LIN {X 0,Y 453.515,Z 483.113,A -85,B 0,C 180,E1 -8409.446,E2 -8409.446} C_VEL
LIN {X 0,Y 453.464,Z 483.111,A -85,B 0,C 180,E1 -8412.994,E2 -8412.994} C_VEL
LIN {X 0,Y 453.46,Z 483.124,A -85,B 0,C 180,E1 -8415.778,E2 -8415.778} C_VEL
LIN {X 0,Y 453.512,Z 483.122,A -85,B 0,C 180,E1 -8419.405,E2 -8419.405} C_VEL
LIN {X 0,Y 453.471,Z 483.115,A -85,B 0,C 180,E1 -8422.222,E2 -8422.222} C_VEL
LIN {X 0,Y 453.484,Z 483.123,A -85,B 0,C 180,E1 -8425.222,E2 -8425.222} C_VEL
LIN {X 0,Y 453.46,Z 483.119,A -85,B 0,C 180,E1 -8428.474,E2 -8428.474} C_VEL
LIN {X 0,Y 453.531,Z 483.104,A -85,B 0,C 180,E1 -8432.038,E2 -8432.038} C_VEL
LIN {X 0,Y 453.507,Z 483.119,A -85,B 0,C 180,E1 -8435.265,E2 -8435.265} C_VEL
LIN {X 0,Y 453.473,Z 483.112,A -85,B 0,C 180,E1 -8438.414,E2 -8438.414} C_VEL
LIN {X 0,Y 453.514,Z 483.11,A -85,B 0,C 180,E1 -8441.008,E2 -8441.008} C_VEL
LIN {X 0,Y 453.561,Z 483.108,A -85,B 0,C 180,E1 -8443.879,E2 -8443.879} C_VEL
LIN {X 0,Y 453.555,Z 483.102,A -85,B 0,C 180,E1 -8447.471,E2 -8447.471} C_VEL
LIN {X 0,Y 453.584,Z 483.109,A -85,B 0,C 180,E1 -8451.086,E2 -8451.086} C_VEL
LIN {X 0,Y 453.669,Z 483.082,A -85,B 0,C 180,E1 -8453.774,E2 -8453.774} C_VEL
LIN {X 0,Y 453.757,Z 483.086,A -85,B 0,C 180,E1 -8457.336,E2 -8457.336} C_VEL
LIN {X 0,Y 453.814,Z 483.072,A -85,B 0,C 180,E1 -8460,E2 -8460} C_VEL
LIN {X 0,Y 453.757,Z 483.069,A -85,B 0,C 180,E1 -8462.663,E2 -8462.663} C_VEL
LIN {X 0,Y 453.667,Z 483.095,A -85,B 0,C 180,E1 -8466.225,E2 -8466.225} C_VEL
LIN {X 0,Y 453.583,Z 483.099,A -85,B 0,C 180,E1 -8468.913,E2 -8468.913} C_VEL
LIN {X 0,Y 453.554,Z 483.108,A -85,B 0,C 180,E1 -8472.529,E2 -8472.529} C_VEL
LIN {X 0,Y 453.535,Z 483.104,A -85,B 0,C 180,E1 -8476.196,E2 -8476.196} C_VEL
LIN {X 0,Y 453.51,Z 483.11,A -85,B 0,C 180,E1 -8479.041,E2 -8479.041} C_VEL
LIN {X 0,Y 453.466,Z 483.122,A -85,B 0,C 180,E1 -8481.836,E2 -8481.836} C_VEL
LIN {X 0,Y 453.504,Z 483.105,A -85,B 0,C 180,E1 -8484.734,E2 -8484.734} C_VEL
LIN {X 0,Y 453.529,Z 483.115,A -85,B 0,C 180,E1 -8487.961,E2 -8487.961} C_VEL
LIN {X 0,Y 453.474,Z 483.109,A -85,B 0,C 180,E1 -8490.759,E2 -8490.759} C_VEL
LIN {X 0,Y 453.469,Z 483.123,A -85,B 0,C 180,E1 -8493.913,E2 -8493.913} C_VEL
LIN {X 0,Y 453.462,Z 483.119,A -85,B 0,C 180,E1 -8497.188,E2 -8497.188} C_VEL
LIN {X 0,Y 453.508,Z 483.121,A -85,B 0,C 180,E1 -8499.447,E2 -8499.447} C_VEL
LIN {X 0,Y 453.484,Z 483.12,A -85,B 0,C 180,E1 -8502.992,E2 -8502.992} C_VEL
LIN {X 0,Y 453.469,Z 483.104,A -85,B 0,C 180,E1 -8505.781,E2 -8505.781} C_VEL
LIN {X 0,Y 453.49,Z 483.109,A -85,B 0,C 180,E1 -8508.212,E2 -8508.212} C_VEL
LIN {X 0,Y 453.528,Z 483.114,A -85,B 0,C 180,E1 -8510.787,E2 -8510.787} C_VEL
LIN {X 0,Y 453.45,Z 483.113,A -85,B 0,C 180,E1 -8513.918,E2 -8513.918} C_VEL
LIN {X 0,Y 453.477,Z 483.122,A -85,B 0,C 180,E1 -8517.152,E2 -8517.152} C_VEL
LIN {X 0,Y 453.508,Z 483.12,A -85,B 0,C 180,E1 -8520.271,E2 -8520.271} C_VEL
LIN {X 0,Y 453.504,Z 483.12,A -85,B 0,C 180,E1 -8523.294,E2 -8523.294} C_VEL
LIN {X 0,Y 453.499,Z 483.122,A -85,B 0,C 180,E1 -8526.239,E2 -8526.239} C_VEL
LIN {X 0,Y 453.478,Z 483.122,A -85,B 0,C 180,E1 -8529.118,E2 -8529.118} C_VEL
LIN {X 0,Y 453.507,Z 483.123,A -85,B 0,C 180,E1 -8531.945,E2 -8531.945} C_VEL
LIN {X 0,Y 453.535,Z 483.116,A -85,B 0,C 180,E1 -8534.727,E2 -8534.727} C_VEL
LIN {X 0,Y 453.556,Z 483.115,A -85,B 0,C 180,E1 -8538.379,E2 -8538.379} C_VEL
LIN {X 0,Y 453.648,Z 483.104,A -85,B 0,C 180,E1 -8541.985,E2 -8541.985} C_VEL
LIN {X 0,Y 453.633,Z 483.102,A -85,B 0,C 180,E1 -8543.101,E2 -8543.101} C_VEL
LIN {X 0,Y 452.948,Z 483.192,A -85,B 0,C 180,E1 -8543.841,E2 -8543.841} C_VEL
LIN {X 0,Y 450,Z 483.556,A -85,B 0,C 180,E1 -8545.043,E2 -8545.043} C_VEL
LIN {X 0,Y 447.578,Z 483.861,A -85,B 0,C 180,E1 -8546.012,E2 -8546.012} C_VEL
LIN {X 0,Y 446.643,Z 483.975,A -85,B 0,C 180,E1 -8546.762,E2 -8546.762} C_VEL
LIN {X 0,Y 446.623,Z 483.977,A -85,B 0,C 180,E1 -8547.016,E2 -8547.016} C_VEL
LIN {X 0,Y 446.791,Z 483.959,A -85,B 0,C 180,E1 -8550,E2 -8550} C_VEL
LIN {X 0,Y 446.706,Z 483.968,A -85,B 0,C 180,E1 -8552.705,E2 -8552.705} C_VEL
LIN {X 0,Y 446.643,Z 483.977,A -85,B 0,C 180,E1 -8556.324,E2 -8556.324} C_VEL
LIN {X 0,Y 446.534,Z 483.987,A -85,B 0,C 180,E1 -8559.055,E2 -8559.055} C_VEL
LIN {X 0,Y 446.517,Z 483.99,A -85,B 0,C 180,E1 -8562.73,E2 -8562.73} C_VEL
LIN {X 0,Y 446.492,Z 483.996,A -85,B 0,C 180,E1 -8566.228,E2 -8566.228} C_VEL
LIN {X 0,Y 446.465,Z 483.997,A -85,B 0,C 180,E1 -8569.303,E2 -8569.303} C_VEL
LIN {X 0,Y 446.414,Z 484.005,A -85,B 0,C 180,E1 -8572.199,E2 -8572.199} C_VEL
LIN {X 0,Y 446.452,Z 483.997,A -85,B 0,C 180,E1 -8575.152,E2 -8575.152} C_VEL
LIN {X 0,Y 446.479,Z 483.998,A -85,B 0,C 180,E1 -8578.178,E2 -8578.178} C_VEL
LIN {X 0,Y 446.414,Z 484.001,A -85,B 0,C 180,E1 -8581.3,E2 -8581.3} C_VEL
LIN {X 0,Y 446.424,Z 484,A -85,B 0,C 180,E1 -8584.523,E2 -8584.523} C_VEL
LIN {X 0,Y 446.431,Z 483.991,A -85,B 0,C 180,E1 -8588.083,E2 -8588.083} C_VEL
LIN {X 0,Y 446.44,Z 483.993,A -85,B 0,C 180,E1 -8590.92,E2 -8590.92} C_VEL
LIN {X 0,Y 446.437,Z 483.973,A -85,B 0,C 180,E1 -8593.84,E2 -8593.84} C_VEL
LIN {X 0,Y 446.439,Z 484.003,A -85,B 0,C 180,E1 -8596.397,E2 -8596.397} C_VEL
LIN {X 0,Y 446.443,Z 483.991,A -85,B 0,C 180,E1 -8599.803,E2 -8599.803} C_VEL
LIN {X 0,Y 446.419,Z 484.005,A -85,B 0,C 180,E1 -8602.123,E2 -8602.123} C_VEL
LIN {X 0,Y 446.421,Z 483.996,A -85,B 0,C 180,E1 -8605.477,E2 -8605.477} C_VEL
LIN {X 0,Y 446.41,Z 483.992,A -85,B 0,C 180,E1 -8608.7,E2 -8608.7} C_VEL
LIN {X 0,Y 446.475,Z 483.992,A -85,B 0,C 180,E1 -8611.821,E2 -8611.821} C_VEL
LIN {X 0,Y 446.448,Z 483.986,A -85,B 0,C 180,E1 -8614.848,E2 -8614.848} C_VEL
LIN {X 0,Y 446.438,Z 483.999,A -85,B 0,C 180,E1 -8618.245,E2 -8618.245} C_VEL
LIN {X 0,Y 446.448,Z 483.988,A -85,B 0,C 180,E1 -8621.649,E2 -8621.649} C_VEL
LIN {X 0,Y 446.498,Z 483.989,A -85,B 0,C 180,E1 -8624.48,E2 -8624.48} C_VEL
LIN {X 0,Y 446.509,Z 483.988,A -85,B 0,C 180,E1 -8628.193,E2 -8628.193} C_VEL
LIN {X 0,Y 446.591,Z 483.97,A -85,B 0,C 180,E1 -8631.858,E2 -8631.858} C_VEL
LIN {X 0,Y 446.643,Z 483.973,A -85,B 0,C 180,E1 -8634.583,E2 -8634.583} C_VEL
LIN {X 0,Y 446.701,Z 483.948,A -85,B 0,C 180,E1 -8637.295,E2 -8637.295} C_VEL
LIN {X 0,Y 446.784,Z 483.947,A -85,B 0,C 180,E1 -8640,E2 -8640} C_VEL
LIN {X 0,Y 446.701,Z 483.964,A -85,B 0,C 180,E1 -8642.706,E2 -8642.706} C_VEL
LIN {X 0,Y 446.638,Z 483.958,A -85,B 0,C 180,E1 -8646.324,E2 -8646.324} C_VEL
LIN {X 0,Y 446.53,Z 483.987,A -85,B 0,C 180,E1 -8649.056,E2 -8649.056} C_VEL
LIN {X 0,Y 446.513,Z 483.976,A -85,B 0,C 180,E1 -8652.73,E2 -8652.73} C_VEL
LIN {X 0,Y 446.482,Z 483.994,A -85,B 0,C 180,E1 -8656.46,E2 -8656.46} C_VEL
LIN {X 0,Y 446.462,Z 483.986,A -85,B 0,C 180,E1 -8659.304,E2 -8659.304} C_VEL
LIN {X 0,Y 446.411,Z 483.994,A -85,B 0,C 180,E1 -8662.2,E2 -8662.2} C_VEL
LIN {X 0,Y 446.451,Z 483.993,A -85,B 0,C 180,E1 -8665.153,E2 -8665.153} C_VEL
LIN {X 0,Y 446.478,Z 483.984,A -85,B 0,C 180,E1 -8668.179,E2 -8668.179} C_VEL
LIN {X 0,Y 446.414,Z 483.997,A -85,B 0,C 180,E1 -8671.776,E2 -8671.776} C_VEL
LIN {X 0,Y 446.425,Z 483.998,A -85,B 0,C 180,E1 -8674.524,E2 -8674.524} C_VEL
LIN {X 0,Y 446.431,Z 483.992,A -85,B 0,C 180,E1 -8678.084,E2 -8678.084} C_VEL
LIN {X 0,Y 446.439,Z 483.998,A -85,B 0,C 180,E1 -8680.921,E2 -8680.921} C_VEL
LIN {X 0,Y 446.396,Z 484.003,A -85,B 0,C 180,E1 -8683.847,E2 -8683.847} C_VEL
LIN {X 0,Y 446.417,Z 483.989,A -85,B 0,C 180,E1 -8686.401,E2 -8686.401} C_VEL
LIN {X 0,Y 446.449,Z 483.996,A -85,B 0,C 180,E1 -8689.804,E2 -8689.804} C_VEL
LIN {X 0,Y 446.407,Z 483.973,A -85,B 0,C 180,E1 -8692.122,E2 -8692.122} C_VEL
LIN {X 0,Y 446.428,Z 483.989,A -85,B 0,C 180,E1 -8695.478,E2 -8695.478} C_VEL
LIN {X 0,Y 446.417,Z 483.974,A -85,B 0,C 180,E1 -8698.701,E2 -8698.701} C_VEL
LIN {X 0,Y 446.476,Z 484.115,A -85,B 0,C 180,E1 -8699.755,E2 -8699.755} C_VEL
LIN {X 0,Y 448.83,Z 495.487,A -85,B 0,C 180,E1 -8702.489,E2 -8702.489} C_VEL
LIN {X 0,Y 449.538,Z 500.19,A -85,B 0,C 180,E1 -8703.541,E2 -8703.541} C_VEL
LIN {X 0,Y 448.777,Z 514.196,A -85,B 0,C 180,E1 -8706.464,E2 -8706.464} C_VEL
LIN {X 0,Y 448.217,Z 523.143,A -85,B 0,C 180,E1 -8708.318,E2 -8708.318} C_VEL
LIN {X 0,Y 449.163,Z 527.943,A -85,B 0,C 180,E1 -8708.491,E2 -8708.491} C_VEL
LIN {X 0,Y 453.386,Z 549.291,A -85,B 0,C 180,E1 -8709.054,E2 -8709.054} C_VEL
LIN {X 0,Y 452.142,Z 657.267,A -85,B 0,C 180,E1 -8710.802,E2 -8710.802} C_VEL
LIN {X 0,Y 451.794,Z 668.666,A -85,B 0,C 180,E1 -8711.081,E2 -8711.081} C_VEL
LIN {X 0,Y 451.343,Z 679.209,A -85,B 0,C 180,E1 -8711.444,E2 -8711.444} C_VEL
LIN {X 0,Y 450.892,Z 689.76,A -85,B 0,C 180,E1 -8711.921,E2 -8711.921} C_VEL
LIN {X 0,Y 450.291,Z 700.274,A -85,B 0,C 180,E1 -8712.511,E2 -8712.511} C_VEL
LIN {X 0,Y 449.69,Z 710.266,A -85,B 0,C 180,E1 -8713.195,E2 -8713.195} C_VEL
LIN {X 0,Y 449.012,Z 719.993,A -85,B 0,C 180,E1 -8713.987,E2 -8713.987} C_VEL
LIN {X 0,Y 448.336,Z 729.416,A -85,B 0,C 180,E1 -8714.894,E2 -8714.894} C_VEL
LIN {X 0,Y 447.671,Z 738.441,A -85,B 0,C 180,E1 -8715.917,E2 -8715.917} C_VEL
LIN {X 0,Y 447.112,Z 746.926,A -85,B 0,C 180,E1 -8717.049,E2 -8717.049} C_VEL
LIN {X 0,Y 446.683,Z 754.285,A -85,B 0,C 180,E1 -8718.198,E2 -8718.198} C_VEL
LIN {X 0,Y 446.237,Z 760.559,A -85,B 0,C 180,E1 -8719.336,E2 -8719.336} C_VEL
LIN {X 0,Y 445.953,Z 765.962,A -85,B 0,C 180,E1 -8720.475,E2 -8720.475} C_VEL
LIN {X 0,Y 445.697,Z 771.394,A -85,B 0,C 180,E1 -8721.841,E2 -8721.841} C_VEL
LIN {X 0,Y 445.57,Z 775.838,A -85,B 0,C 180,E1 -8723.207,E2 -8723.207} C_VEL
LIN {X 0,Y 445.476,Z 779.378,A -85,B 0,C 180,E1 -8724.568,E2 -8724.568} C_VEL
LIN {X 0,Y 445.395,Z 781.314,A -85,B 0,C 180,E1 -8725.475,E2 -8725.475} C_VEL
LIN {X 0,Y 445.429,Z 783.994,A -85,B 0,C 180,E1 -8727.287,E2 -8727.287} C_VEL
LIN {X 0,Y 445.336,Z 785.278,A -85,B 0,C 180,E1 -8729.096,E2 -8729.096} C_VEL
LIN {X 0,Y 445.341,Z 785.529,A -85,B 0,C 180,E1 -8730,E2 -8730} C_VEL
LIN {X 0,Y 445.353,Z 784.807,A -85,B 0,C 180,E1 -8731.809,E2 -8731.809} C_VEL
LIN {X 0,Y 445.429,Z 783.994,A -85,B 0,C 180,E1 -8732.713,E2 -8732.713} C_VEL
LIN {X 0,Y 445.395,Z 781.314,A -85,B 0,C 180,E1 -8734.525,E2 -8734.525} C_VEL
LIN {X 0,Y 445.529,Z 776.974,A -85,B 0,C 180,E1 -8736.385,E2 -8736.385} C_VEL
LIN {X 0,Y 445.621,Z 772.972,A -85,B 0,C 180,E1 -8737.704,E2 -8737.704} C_VEL
LIN {X 0,Y 445.884,Z 767.876,A -85,B 0,C 180,E1 -8739.069,E2 -8739.069} C_VEL
LIN {X 0,Y 446.179,Z 761.697,A -85,B 0,C 180,E1 -8740.436,E2 -8740.436} C_VEL
LIN {X 0,Y 446.605,Z 755.623,A -85,B 0,C 180,E1 -8741.574,E2 -8741.574} C_VEL
LIN {X 0,Y 447.018,Z 748.545,A -85,B 0,C 180,E1 -8742.715,E2 -8742.715} C_VEL
LIN {X 0,Y 447.442,Z 742.08,A -85,B 0,C 180,E1 -8743.627,E2 -8743.627} C_VEL
LIN {X 0,Y 448.128,Z 732.597,A -85,B 0,C 180,E1 -8744.764,E2 -8744.764} C_VEL
LIN {X 0,Y 448.713,Z 723.714,A -85,B 0,C 180,E1 -8745.675,E2 -8745.675} C_VEL
LIN {X 0,Y 449.406,Z 714.661,A -85,B 0,C 180,E1 -8746.466,E2 -8746.466} C_VEL
LIN {X 0,Y 450.11,Z 703.851,A -85,B 0,C 180,E1 -8747.257,E2 -8747.257} C_VEL
LIN {X 0,Y 450.666,Z 694.13,A -85,B 0,C 180,E1 -8747.85,E2 -8747.85} C_VEL
LIN {X 0,Y 451.166,Z 683.291,A -85,B 0,C 180,E1 -8748.387,E2 -8748.387} C_VEL
LIN {X 0,Y 451.69,Z 671.402,A -85,B 0,C 180,E1 -8748.835,E2 -8748.835} C_VEL
LIN {X 0,Y 452.062,Z 659.986,A -85,B 0,C 180,E1 -8749.143,E2 -8749.143} C_VEL
LIN {X 0,Y 452.545,Z 631.666,A -85,B 0,C 180,E1 -8749.623,E2 -8749.623} C_VEL
LIN {X 0,Y 453.344,Z 548.908,A -85,B 0,C 180,E1 -8750.955,E2 -8750.955} C_VEL
LIN {X 0,Y 448.23,Z 523.43,A -85,B 0,C 180,E1 -8751.653,E2 -8751.653} C_VEL
LIN {X 0,Y 448.295,Z 522.142,A -85,B 0,C 180,E1 -8751.859,E2 -8751.859} C_VEL
LIN {X 0,Y 449.213,Z 507.408,A -85,B 0,C 180,E1 -8754.987,E2 -8754.987} C_VEL
LIN {X 0,Y 449.593,Z 500.365,A -85,B 0,C 180,E1 -8756.455,E2 -8756.455} C_VEL
LIN {X 0,Y 448.145,Z 491.791,A -85,B 0,C 180,E1 -8758.378,E2 -8758.378} C_VEL
LIN {X 0,Y 446.476,Z 484.118,A -85,B 0,C 180,E1 -8760.245,E2 -8760.245} C_VEL
LIN {X 0,Y 446.444,Z 484.003,A -85,B 0,C 180,E1 -8763.453,E2 -8763.453} C_VEL
LIN {X 0,Y 446.399,Z 483.96,A -85,B 0,C 180,E1 -8766.745,E2 -8766.745} C_VEL
LIN {X 0,Y 446.476,Z 483.991,A -85,B 0,C 180,E1 -8769.528,E2 -8769.528} C_VEL
LIN {X 0,Y 446.429,Z 483.99,A -85,B 0,C 180,E1 -8772.603,E2 -8772.603} C_VEL
LIN {X 0,Y 446.45,Z 483.993,A -85,B 0,C 180,E1 -8775.103,E2 -8775.103} C_VEL
LIN {X 0,Y 446.431,Z 483.994,A -85,B 0,C 180,E1 -8778.609,E2 -8778.609} C_VEL
LIN {X 0,Y 446.468,Z 483.997,A -85,B 0,C 180,E1 -8780.975,E2 -8780.975} C_VEL
LIN {X 0,Y 446.416,Z 483.999,A -85,B 0,C 180,E1 -8784.373,E2 -8784.373} C_VEL
LIN {X 0,Y 446.417,Z 483.998,A -85,B 0,C 180,E1 -8787.638,E2 -8787.638} C_VEL
LIN {X 0,Y 446.443,Z 483.997,A -85,B 0,C 180,E1 -8790.79,E2 -8790.79} C_VEL
LIN {X 0,Y 446.471,Z 483.991,A -85,B 0,C 180,E1 -8793.848,E2 -8793.848} C_VEL
LIN {X 0,Y 446.422,Z 483.999,A -85,B 0,C 180,E1 -8796.823,E2 -8796.823} C_VEL
LIN {X 0,Y 446.437,Z 483.989,A -85,B 0,C 180,E1 -8799.736,E2 -8799.736} C_VEL
LIN {X 0,Y 446.456,Z 483.994,A -85,B 0,C 180,E1 -8802.596,E2 -8802.596} C_VEL
LIN {X 0,Y 446.461,Z 483.986,A -85,B 0,C 180,E1 -8805.412,E2 -8805.412} C_VEL
LIN {X 0,Y 446.509,Z 483.984,A -85,B 0,C 180,E1 -8808.192,E2 -8808.192} C_VEL
LIN {X 0,Y 446.592,Z 483.975,A -85,B 0,C 180,E1 -8811.857,E2 -8811.857} C_VEL
LIN {X 0,Y 446.637,Z 483.954,A -85,B 0,C 180,E1 -8814.582,E2 -8814.582} C_VEL
LIN {X 0,Y 446.701,Z 483.964,A -85,B 0,C 180,E1 -8817.294,E2 -8817.294} C_VEL
LIN {X 0,Y 446.784,Z 483.947,A -85,B 0,C 180,E1 -8820,E2 -8820} C_VEL
LIN {X 0,Y 446.701,Z 483.948,A -85,B 0,C 180,E1 -8822.705,E2 -8822.705} C_VEL
LIN {X 0,Y 446.637,Z 483.97,A -85,B 0,C 180,E1 -8826.323,E2 -8826.323} C_VEL
LIN {X 0,Y 446.529,Z 483.978,A -85,B 0,C 180,E1 -8829.055,E2 -8829.055} C_VEL
LIN {X 0,Y 446.512,Z 483.986,A -85,B 0,C 180,E1 -8832.73,E2 -8832.73} C_VEL
LIN {X 0,Y 446.486,Z 483.981,A -85,B 0,C 180,E1 -8836.228,E2 -8836.228} C_VEL
LIN {X 0,Y 446.46,Z 483.99,A -85,B 0,C 180,E1 -8839.303,E2 -8839.303} C_VEL
LIN {X 0,Y 446.408,Z 483.998,A -85,B 0,C 180,E1 -8842.2,E2 -8842.2} C_VEL
LIN {X 0,Y 446.448,Z 483.986,A -85,B 0,C 180,E1 -8845.152,E2 -8845.152} C_VEL
LIN {X 0,Y 446.475,Z 483.992,A -85,B 0,C 180,E1 -8848.179,E2 -8848.179} C_VEL
LIN {X 0,Y 446.41,Z 483.992,A -85,B 0,C 180,E1 -8851.3,E2 -8851.3} C_VEL
LIN {X 0,Y 446.421,Z 483.996,A -85,B 0,C 180,E1 -8854.523,E2 -8854.523} C_VEL
LIN {X 0,Y 446.422,Z 484.002,A -85,B 0,C 180,E1 -8858.082,E2 -8858.082} C_VEL
LIN {X 0,Y 446.422,Z 483.991,A -85,B 0,C 180,E1 -8860.918,E2 -8860.918} C_VEL
LIN {X 0,Y 446.437,Z 483.999,A -85,B 0,C 180,E1 -8863.841,E2 -8863.841} C_VEL
LIN {X 0,Y 446.439,Z 483.97,A -85,B 0,C 180,E1 -8866.397,E2 -8866.397} C_VEL
LIN {X 0,Y 446.463,Z 483.998,A -85,B 0,C 180,E1 -8869.805,E2 -8869.805} C_VEL
LIN {X 0,Y 446.428,Z 483.989,A -85,B 0,C 180,E1 -8872.124,E2 -8872.124} C_VEL
LIN {X 0,Y 446.424,Z 484,A -85,B 0,C 180,E1 -8875.477,E2 -8875.477} C_VEL
LIN {X 0,Y 446.414,Z 484.001,A -85,B 0,C 180,E1 -8878.7,E2 -8878.7} C_VEL
LIN {X 0,Y 446.479,Z 483.998,A -85,B 0,C 180,E1 -8881.822,E2 -8881.822} C_VEL
LIN {X 0,Y 446.452,Z 483.997,A -85,B 0,C 180,E1 -8884.848,E2 -8884.848} C_VEL
LIN {X 0,Y 446.443,Z 484.001,A -85,B 0,C 180,E1 -8888.245,E2 -8888.245} C_VEL
LIN {X 0,Y 446.453,Z 484,A -85,B 0,C 180,E1 -8891.649,E2 -8891.649} C_VEL
LIN {X 0,Y 446.503,Z 483.993,A -85,B 0,C 180,E1 -8894.48,E2 -8894.48} C_VEL
LIN {X 0,Y 446.514,Z 483.993,A -85,B 0,C 180,E1 -8898.193,E2 -8898.193} C_VEL
LIN {X 0,Y 446.596,Z 483.982,A -85,B 0,C 180,E1 -8901.858,E2 -8901.858} C_VEL
LIN {X 0,Y 446.642,Z 483.975,A -85,B 0,C 180,E1 -8904.583,E2 -8904.583} C_VEL
LIN {X 0,Y 446.623,Z 483.977,A -85,B 0,C 180,E1 -8907.016,E2 -8907.016} C_VEL
LIN {X 0,Y 446.106,Z 484.044,A -85,B 0,C 180,E1 -8907.769,E2 -8907.769} C_VEL
LIN {X 0,Y 443.288,Z 484.397,A -85,B 0,C 180,E1 -8908.992,E2 -8908.992} C_VEL
LIN {X 0,Y 440.8,Z 484.706,A -85,B 0,C 180,E1 -8909.979,E2 -8909.979} C_VEL
LIN {X 0,Y 439.712,Z 484.84,A -85,B 0,C 180,E1 -8910.742,E2 -8910.742} C_VEL
LIN {X 0,Y 439.618,Z 484.85,A -85,B 0,C 180,E1 -8911.001,E2 -8911.001} C_VEL
LIN {X 0,Y 439.652,Z 484.847,A -85,B 0,C 180,E1 -8912.749,E2 -8912.749} C_VEL
LIN {X 0,Y 439.614,Z 484.852,A -85,B 0,C 180,E1 -8916.425,E2 -8916.425} C_VEL
LIN {X 0,Y 439.496,Z 484.864,A -85,B 0,C 180,E1 -8919.201,E2 -8919.201} C_VEL
LIN {X 0,Y 439.461,Z 484.869,A -85,B 0,C 180,E1 -8922.937,E2 -8922.937} C_VEL
LIN {X 0,Y 439.443,Z 484.873,A -85,B 0,C 180,E1 -8926.349,E2 -8926.349} C_VEL
LIN {X 0,Y 439.398,Z 484.878,A -85,B 0,C 180,E1 -8929.626,E2 -8929.626} C_VEL
LIN {X 0,Y 439.361,Z 484.882,A -85,B 0,C 180,E1 -8932.575,E2 -8932.575} C_VEL
LIN {X 0,Y 439.4,Z 484.878,A -85,B 0,C 180,E1 -8935.585,E2 -8935.585} C_VEL
LIN {X 0,Y 439.419,Z 484.875,A -85,B 0,C 180,E1 -8938.673,E2 -8938.673} C_VEL
LIN {X 0,Y 439.369,Z 484.883,A -85,B 0,C 180,E1 -8941.86,E2 -8941.86} C_VEL
LIN {X 0,Y 439.394,Z 484.872,A -85,B 0,C 180,E1 -8945.155,E2 -8945.155} C_VEL
LIN {X 0,Y 439.393,Z 484.877,A -85,B 0,C 180,E1 -8948.593,E2 -8948.593} C_VEL
LIN {X 0,Y 439.397,Z 484.869,A -85,B 0,C 180,E1 -8951.259,E2 -8951.259} C_VEL
LIN {X 0,Y 439.402,Z 484.865,A -85,B 0,C 180,E1 -8954.728,E2 -8954.728} C_VEL
LIN {X 0,Y 439.403,Z 484.876,A -85,B 0,C 180,E1 -8957.797,E2 -8957.797} C_VEL
LIN {X 0,Y 439.428,Z 484.87,A -85,B 0,C 180,E1 -8960.228,E2 -8960.228} C_VEL
LIN {X 0,Y 439.368,Z 484.874,A -85,B 0,C 180,E1 -8963.713,E2 -8963.713} C_VEL
LIN {X 0,Y 439.366,Z 484.877,A -85,B 0,C 180,E1 -8967.054,E2 -8967.054} C_VEL
LIN {X 0,Y 439.387,Z 484.869,A -85,B 0,C 180,E1 -8970.275,E2 -8970.275} C_VEL
LIN {X 0,Y 439.424,Z 484.869,A -85,B 0,C 180,E1 -8973.589,E2 -8973.589} C_VEL
LIN {X 0,Y 439.377,Z 484.869,A -85,B 0,C 180,E1 -8976.43,E2 -8976.43} C_VEL
LIN {X 0,Y 439.379,Z 484.875,A -85,B 0,C 180,E1 -8979.397,E2 -8979.397} C_VEL
LIN {X 0,Y 439.422,Z 484.861,A -85,B 0,C 180,E1 -8982.31,E2 -8982.31} C_VEL
LIN {X 0,Y 439.437,Z 484.868,A -85,B 0,C 180,E1 -8985.174,E2 -8985.174} C_VEL
LIN {X 0,Y 439.475,Z 484.865,A -85,B 0,C 180,E1 -8988.002,E2 -8988.002} C_VEL
LIN {X 0,Y 439.539,Z 484.847,A -85,B 0,C 180,E1 -8991.727,E2 -8991.727} C_VEL
LIN {X 0,Y 439.618,Z 484.85,A -85,B 0,C 180,E1 -8994.496,E2 -8994.496} C_VEL
LIN {X 0,Y 439.627,Z 484.83,A -85,B 0,C 180,E1 -8998.168,E2 -8998.168} C_VEL
LIN {X 0,Y 439.754,Z 484.823,A -85,B 0,C 180,E1 -9000,E2 -9000} C_VEL
LIN {X 0,Y 439.648,Z 484.842,A -85,B 0,C 180,E1 -9002.749,E2 -9002.749} C_VEL
LIN {X 0,Y 439.609,Z 484.834,A -85,B 0,C 180,E1 -9006.426,E2 -9006.426} C_VEL
LIN {X 0,Y 439.492,Z 484.862,A -85,B 0,C 180,E1 -9009.202,E2 -9009.202} C_VEL
LIN {X 0,Y 439.458,Z 484.852,A -85,B 0,C 180,E1 -9012.938,E2 -9012.938} C_VEL
LIN {X 0,Y 439.439,Z 484.869,A -85,B 0,C 180,E1 -9016.349,E2 -9016.349} C_VEL
LIN {X 0,Y 439.395,Z 484.866,A -85,B 0,C 180,E1 -9019.627,E2 -9019.627} C_VEL
LIN {X 0,Y 439.358,Z 484.878,A -85,B 0,C 180,E1 -9022.576,E2 -9022.576} C_VEL
LIN {X 0,Y 439.399,Z 484.869,A -85,B 0,C 180,E1 -9025.586,E2 -9025.586} C_VEL
LIN {X 0,Y 439.411,Z 484.871,A -85,B 0,C 180,E1 -9028.674,E2 -9028.674} C_VEL
LIN {X 0,Y 439.365,Z 484.876,A -85,B 0,C 180,E1 -9032.031,E2 -9032.031} C_VEL
LIN {X 0,Y 439.391,Z 484.875,A -85,B 0,C 180,E1 -9035.342,E2 -9035.342} C_VEL
LIN {X 0,Y 439.392,Z 484.873,A -85,B 0,C 180,E1 -9038.594,E2 -9038.594} C_VEL
LIN {X 0,Y 439.394,Z 484.872,A -85,B 0,C 180,E1 -9041.259,E2 -9041.259} C_VEL
LIN {X 0,Y 439.398,Z 484.875,A -85,B 0,C 180,E1 -9044.73,E2 -9044.73} C_VEL
LIN {X 0,Y 439.395,Z 484.868,A -85,B 0,C 180,E1 -9047.797,E2 -9047.797} C_VEL
LIN {X 0,Y 439.434,Z 484.872,A -85,B 0,C 180,E1 -9050.229,E2 -9050.229} C_VEL
LIN {X 0,Y 439.371,Z 484.834,A -85,B 0,C 180,E1 -9053.714,E2 -9053.714} C_VEL
LIN {X 0,Y 439.372,Z 484.878,A -85,B 0,C 180,E1 -9057.055,E2 -9057.055} C_VEL
LIN {X 0,Y 439.439,Z 484.948,A -85,B 0,C 180,E1 -9059.442,E2 -9059.442} C_VEL
LIN {X 0,Y 441.81,Z 496.456,A -85,B 0,C 180,E1 -9062.272,E2 -9062.272} C_VEL
LIN {X 0,Y 442.632,Z 502.334,A -85,B 0,C 180,E1 -9063.604,E2 -9063.604} C_VEL
LIN {X 0,Y 441.67,Z 517.613,A -85,B 0,C 180,E1 -9066.832,E2 -9066.832} C_VEL
LIN {X 0,Y 441.34,Z 522.992,A -85,B 0,C 180,E1 -9067.97,E2 -9067.97} C_VEL
LIN {X 0,Y 442.627,Z 529.447,A -85,B 0,C 180,E1 -9068.186,E2 -9068.186} C_VEL
LIN {X 0,Y 446.778,Z 550.731,A -85,B 0,C 180,E1 -9068.757,E2 -9068.757} C_VEL
LIN {X 0,Y 445.406,Z 658.429,A -85,B 0,C 180,E1 -9070.53,E2 -9070.53} C_VEL
LIN {X 0,Y 445.047,Z 669.38,A -85,B 0,C 180,E1 -9070.813,E2 -9070.813} C_VEL
LIN {X 0,Y 444.546,Z 680.371,A -85,B 0,C 180,E1 -9071.209,E2 -9071.209} C_VEL
LIN {X 0,Y 444.096,Z 690.242,A -85,B 0,C 180,E1 -9071.672,E2 -9071.672} C_VEL
LIN {X 0,Y 443.489,Z 700.483,A -85,B 0,C 180,E1 -9072.262,E2 -9072.262} C_VEL
LIN {X 0,Y 442.848,Z 710.066,A -85,B 0,C 180,E1 -9072.927,E2 -9072.927} C_VEL
LIN {X 0,Y 442.164,Z 719.794,A -85,B 0,C 180,E1 -9073.732,E2 -9073.732} C_VEL
LIN {X 0,Y 441.467,Z 729.217,A -85,B 0,C 180,E1 -9074.653,E2 -9074.653} C_VEL
LIN {X 0,Y 440.753,Z 738.242,A -85,B 0,C 180,E1 -9075.691,E2 -9075.691} C_VEL
LIN {X 0,Y 440.186,Z 746.275,A -85,B 0,C 180,E1 -9076.773,E2 -9076.773} C_VEL
LIN {X 0,Y 439.668,Z 754.085,A -85,B 0,C 180,E1 -9078.007,E2 -9078.007} C_VEL
LIN {X 0,Y 439.232,Z 760.36,A -85,B 0,C 180,E1 -9079.164,E2 -9079.164} C_VEL
LIN {X 0,Y 438.91,Z 765.763,A -85,B 0,C 180,E1 -9080.321,E2 -9080.321} C_VEL
LIN {X 0,Y 438.631,Z 771.195,A -85,B 0,C 180,E1 -9081.709,E2 -9081.709} C_VEL
LIN {X 0,Y 438.496,Z 775.638,A -85,B 0,C 180,E1 -9083.096,E2 -9083.096} C_VEL
LIN {X 0,Y 438.376,Z 779.179,A -85,B 0,C 180,E1 -9084.48,E2 -9084.48} C_VEL
LIN {X 0,Y 438.32,Z 781.116,A -85,B 0,C 180,E1 -9085.402,E2 -9085.402} C_VEL
LIN {X 0,Y 438.337,Z 783.796,A -85,B 0,C 180,E1 -9087.243,E2 -9087.243} C_VEL
LIN {X 0,Y 438.25,Z 785.08,A -85,B 0,C 180,E1 -9089.081,E2 -9089.081} C_VEL
LIN {X 0,Y 438.252,Z 785.332,A -85,B 0,C 180,E1 -9090,E2 -9090} C_VEL
LIN {X 0,Y 438.276,Z 784.609,A -85,B 0,C 180,E1 -9091.838,E2 -9091.838} C_VEL
LIN {X 0,Y 438.337,Z 783.796,A -85,B 0,C 180,E1 -9092.757,E2 -9092.757} C_VEL
LIN {X 0,Y 438.32,Z 781.116,A -85,B 0,C 180,E1 -9094.598,E2 -9094.598} C_VEL
LIN {X 0,Y 438.448,Z 776.903,A -85,B 0,C 180,E1 -9096.442,E2 -9096.442} C_VEL
LIN {X 0,Y 438.542,Z 772.772,A -85,B 0,C 180,E1 -9097.829,E2 -9097.829} C_VEL
LIN {X 0,Y 438.81,Z 767.676,A -85,B 0,C 180,E1 -9099.216,E2 -9099.216} C_VEL
LIN {X 0,Y 439.131,Z 761.497,A -85,B 0,C 180,E1 -9100.605,E2 -9100.605} C_VEL
LIN {X 0,Y 439.596,Z 755.424,A -85,B 0,C 180,E1 -9101.761,E2 -9101.761} C_VEL
LIN {X 0,Y 440.008,Z 748.344,A -85,B 0,C 180,E1 -9102.921,E2 -9102.921} C_VEL
LIN {X 0,Y 440.6,Z 740.061,A -85,B 0,C 180,E1 -9104.078,E2 -9104.078} C_VEL
LIN {X 0,Y 441.243,Z 731.336,A -85,B 0,C 180,E1 -9105.118,E2 -9105.118} C_VEL
LIN {X 0,Y 441.919,Z 722.274,A -85,B 0,C 180,E1 -9106.04,E2 -9106.04} C_VEL
LIN {X 0,Y 442.681,Z 712.997,A -85,B 0,C 180,E1 -9106.842,E2 -9106.842} C_VEL
LIN {X 0,Y 443.296,Z 703.652,A -85,B 0,C 180,E1 -9107.531,E2 -9107.531} C_VEL
LIN {X 0,Y 443.972,Z 692.047,A -85,B 0,C 180,E1 -9108.233,E2 -9108.233} C_VEL
LIN {X 0,Y 444.478,Z 681.732,A -85,B 0,C 180,E1 -9108.734,E2 -9108.734} C_VEL
LIN {X 0,Y 444.995,Z 671.205,A -85,B 0,C 180,E1 -9109.13,E2 -9109.13} C_VEL
LIN {X 0,Y 445.372,Z 659.788,A -85,B 0,C 180,E1 -9109.442,E2 -9109.442} C_VEL
LIN {X 0,Y 445.873,Z 631.468,A -85,B 0,C 180,E1 -9109.929,E2 -9109.929} C_VEL
LIN {X 0,Y 446.646,Z 549.536,A -85,B 0,C 180,E1 -9111.27,E2 -9111.27} C_VEL
LIN {X 0,Y 441.382,Z 523.232,A -85,B 0,C 180,E1 -9112.006,E2 -9112.006} C_VEL
LIN {X 0,Y 441.398,Z 521.932,A -85,B 0,C 180,E1 -9112.219,E2 -9112.219} C_VEL
LIN {X 0,Y 442.263,Z 508.74,A -85,B 0,C 180,E1 -9115.07,E2 -9115.07} C_VEL
LIN {X 0,Y 442.617,Z 500.83,A -85,B 0,C 180,E1 -9116.768,E2 -9116.768} C_VEL
LIN {X 0,Y 440.638,Z 490.592,A -85,B 0,C 180,E1 -9119.136,E2 -9119.136} C_VEL
LIN {X 0,Y 439.439,Z 484.959,A -85,B 0,C 180,E1 -9120.558,E2 -9120.558} C_VEL
LIN {X 0,Y 439.386,Z 484.878,A -85,B 0,C 180,E1 -9124.043,E2 -9124.043} C_VEL
LIN {X 0,Y 439.346,Z 484.837,A -85,B 0,C 180,E1 -9126.886,E2 -9126.886} C_VEL
LIN {X 0,Y 439.411,Z 484.874,A -85,B 0,C 180,E1 -9129.85,E2 -9129.85} C_VEL
LIN {X 0,Y 439.382,Z 484.866,A -85,B 0,C 180,E1 -9132.627,E2 -9132.627} C_VEL
LIN {X 0,Y 439.398,Z 484.874,A -85,B 0,C 180,E1 -9135.27,E2 -9135.27} C_VEL
LIN {X 0,Y 439.394,Z 484.871,A -85,B 0,C 180,E1 -9138.741,E2 -9138.741} C_VEL
LIN {X 0,Y 439.386,Z 484.871,A -85,B 0,C 180,E1 -9141.604,E2 -9141.604} C_VEL
LIN {X 0,Y 439.396,Z 484.876,A -85,B 0,C 180,E1 -9144.843,E2 -9144.843} C_VEL
LIN {X 0,Y 439.367,Z 484.875,A -85,B 0,C 180,E1 -9148.139,E2 -9148.139} C_VEL
LIN {X 0,Y 439.426,Z 484.865,A -85,B 0,C 180,E1 -9151.597,E2 -9151.597} C_VEL
LIN {X 0,Y 439.399,Z 484.869,A -85,B 0,C 180,E1 -9154.414,E2 -9154.414} C_VEL
LIN {X 0,Y 439.358,Z 484.878,A -85,B 0,C 180,E1 -9157.424,E2 -9157.424} C_VEL
LIN {X 0,Y 439.434,Z 484.861,A -85,B 0,C 180,E1 -9160.662,E2 -9160.662} C_VEL
LIN {X 0,Y 439.454,Z 484.863,A -85,B 0,C 180,E1 -9164.224,E2 -9164.224} C_VEL
LIN {X 0,Y 439.475,Z 484.861,A -85,B 0,C 180,E1 -9168.001,E2 -9168.001} C_VEL
LIN {X 0,Y 439.539,Z 484.854,A -85,B 0,C 180,E1 -9171.726,E2 -9171.726} C_VEL
LIN {X 0,Y 439.613,Z 484.829,A -85,B 0,C 180,E1 -9174.495,E2 -9174.495} C_VEL
LIN {X 0,Y 439.627,Z 484.844,A -85,B 0,C 180,E1 -9178.167,E2 -9178.167} C_VEL
LIN {X 0,Y 439.754,Z 484.823,A -85,B 0,C 180,E1 -9180,E2 -9180} C_VEL
LIN {X 0,Y 439.648,Z 484.826,A -85,B 0,C 180,E1 -9182.748,E2 -9182.748} C_VEL
LIN {X 0,Y 439.608,Z 484.845,A -85,B 0,C 180,E1 -9186.425,E2 -9186.425} C_VEL
LIN {X 0,Y 439.491,Z 484.853,A -85,B 0,C 180,E1 -9189.201,E2 -9189.201} C_VEL
LIN {X 0,Y 439.456,Z 484.865,A -85,B 0,C 180,E1 -9192.937,E2 -9192.937} C_VEL
LIN {X 0,Y 439.438,Z 484.859,A -85,B 0,C 180,E1 -9196.349,E2 -9196.349} C_VEL
LIN {X 0,Y 439.393,Z 484.875,A -85,B 0,C 180,E1 -9199.626,E2 -9199.626} C_VEL
LIN {X 0,Y 439.355,Z 484.875,A -85,B 0,C 180,E1 -9202.575,E2 -9202.575} C_VEL
LIN {X 0,Y 439.396,Z 484.869,A -85,B 0,C 180,E1 -9205.585,E2 -9205.585} C_VEL
LIN {X 0,Y 439.416,Z 484.869,A -85,B 0,C 180,E1 -9208.673,E2 -9208.673} C_VEL
LIN {X 0,Y 439.374,Z 484.879,A -85,B 0,C 180,E1 -9212.033,E2 -9212.033} C_VEL
LIN {X 0,Y 439.387,Z 484.874,A -85,B 0,C 180,E1 -9215.341,E2 -9215.341} C_VEL
LIN {X 0,Y 439.382,Z 484.876,A -85,B 0,C 180,E1 -9218.594,E2 -9218.594} C_VEL
LIN {X 0,Y 439.386,Z 484.869,A -85,B 0,C 180,E1 -9221.258,E2 -9221.258} C_VEL
LIN {X 0,Y 439.402,Z 484.868,A -85,B 0,C 180,E1 -9224.728,E2 -9224.728} C_VEL
LIN {X 0,Y 439.405,Z 484.852,A -85,B 0,C 180,E1 -9227.798,E2 -9227.798} C_VEL
LIN {X 0,Y 439.447,Z 484.871,A -85,B 0,C 180,E1 -9230.231,E2 -9230.231} C_VEL
LIN {X 0,Y 439.37,Z 484.863,A -85,B 0,C 180,E1 -9233.713,E2 -9233.713} C_VEL
LIN {X 0,Y 439.366,Z 484.88,A -85,B 0,C 180,E1 -9237.054,E2 -9237.054} C_VEL
LIN {X 0,Y 439.391,Z 484.879,A -85,B 0,C 180,E1 -9240.276,E2 -9240.276} C_VEL
LIN {X 0,Y 439.428,Z 484.875,A -85,B 0,C 180,E1 -9243.589,E2 -9243.589} C_VEL
LIN {X 0,Y 439.382,Z 484.879,A -85,B 0,C 180,E1 -9246.43,E2 -9246.43} C_VEL
LIN {X 0,Y 439.384,Z 484.88,A -85,B 0,C 180,E1 -9249.397,E2 -9249.397} C_VEL
LIN {X 0,Y 439.427,Z 484.875,A -85,B 0,C 180,E1 -9252.31,E2 -9252.31} C_VEL
LIN {X 0,Y 439.443,Z 484.872,A -85,B 0,C 180,E1 -9255.174,E2 -9255.174} C_VEL
LIN {X 0,Y 439.479,Z 484.869,A -85,B 0,C 180,E1 -9258.001,E2 -9258.001} C_VEL
LIN {X 0,Y 439.544,Z 484.861,A -85,B 0,C 180,E1 -9261.726,E2 -9261.726} C_VEL
LIN {X 0,Y 439.617,Z 484.851,A -85,B 0,C 180,E1 -9264.496,E2 -9264.496} C_VEL
LIN {X 0,Y 439.632,Z 484.85,A -85,B 0,C 180,E1 -9268.168,E2 -9268.168} C_VEL
LIN {X 0,Y 439.76,Z 484.835,A -85,B 0,C 180,E1 -9270,E2 -9270} C_VEL
LIN {X 0,Y 439.618,Z 484.85,A -85,B 0,C 180,E1 -9271.001,E2 -9271.001} C_VEL
LIN {X 0,Y 438.902,Z 484.941,A -85,B 0,C 180,E1 -9271.765,E2 -9271.765} C_VEL
LIN {X 0,Y 435.924,Z 485.311,A -85,B 0,C 180,E1 -9273.004,E2 -9273.004} C_VEL
LIN {X 0,Y 433.473,Z 485.617,A -85,B 0,C 180,E1 -9274.004,E2 -9274.004} C_VEL
LIN {X 0,Y 432.5,Z 485.738,A -85,B 0,C 180,E1 -9274.779,E2 -9274.779} C_VEL
LIN {X 0,Y 432.463,Z 485.741,A -85,B 0,C 180,E1 -9275.041,E2 -9275.041} C_VEL
LIN {X 0,Y 432.582,Z 485.729,A -85,B 0,C 180,E1 -9277.679,E2 -9277.679} C_VEL
LIN {X 0,Y 432.388,Z 485.75,A -85,B 0,C 180,E1 -9281.247,E2 -9281.247} C_VEL
LIN {X 0,Y 432.369,Z 485.755,A -85,B 0,C 180,E1 -9284.112,E2 -9284.112} C_VEL
LIN {X 0,Y 432.393,Z 485.75,A -85,B 0,C 180,E1 -9287.011,E2 -9287.011} C_VEL
LIN {X 0,Y 432.334,Z 485.76,A -85,B 0,C 180,E1 -9289.96,E2 -9289.96} C_VEL
LIN {X 0,Y 432.315,Z 485.759,A -85,B 0,C 180,E1 -9292.964,E2 -9292.964} C_VEL
LIN {X 0,Y 432.359,Z 485.756,A -85,B 0,C 180,E1 -9296.032,E2 -9296.032} C_VEL
LIN {X 0,Y 432.347,Z 485.754,A -85,B 0,C 180,E1 -9299.186,E2 -9299.186} C_VEL
LIN {X 0,Y 432.32,Z 485.762,A -85,B 0,C 180,E1 -9302.293,E2 -9302.293} C_VEL
LIN {X 0,Y 432.334,Z 485.754,A -85,B 0,C 180,E1 -9304.677,E2 -9304.677} C_VEL
LIN {X 0,Y 432.346,Z 485.745,A -85,B 0,C 180,E1 -9308.148,E2 -9308.148} C_VEL
LIN {X 0,Y 432.366,Z 485.741,A -85,B 0,C 180,E1 -9311.608,E2 -9311.608} C_VEL
LIN {X 0,Y 432.371,Z 485.731,A -85,B 0,C 180,E1 -9314.341,E2 -9314.341} C_VEL
LIN {X 0,Y 432.358,Z 485.752,A -85,B 0,C 180,E1 -9317.009,E2 -9317.009} C_VEL
LIN {X 0,Y 432.334,Z 485.748,A -85,B 0,C 180,E1 -9319.819,E2 -9319.819} C_VEL
LIN {X 0,Y 432.307,Z 485.752,A -85,B 0,C 180,E1 -9323.023,E2 -9323.023} C_VEL
LIN {X 0,Y 432.351,Z 485.753,A -85,B 0,C 180,E1 -9325.996,E2 -9325.996} C_VEL
LIN {X 0,Y 432.386,Z 485.736,A -85,B 0,C 180,E1 -9329.744,E2 -9329.744} C_VEL
LIN {X 0,Y 432.391,Z 485.745,A -85,B 0,C 180,E1 -9333.372,E2 -9333.372} C_VEL
LIN {X 0,Y 432.362,Z 485.739,A -85,B 0,C 180,E1 -9336.023,E2 -9336.023} C_VEL
LIN {X 0,Y 432.34,Z 485.753,A -85,B 0,C 180,E1 -9339.046,E2 -9339.046} C_VEL
LIN {X 0,Y 432.368,Z 485.741,A -85,B 0,C 180,E1 -9342.011,E2 -9342.011} C_VEL
LIN {X 0,Y 432.385,Z 485.748,A -85,B 0,C 180,E1 -9344.927,E2 -9344.927} C_VEL
LIN {X 0,Y 432.45,Z 485.738,A -85,B 0,C 180,E1 -9347.804,E2 -9347.804} C_VEL
LIN {X 0,Y 432.483,Z 485.726,A -85,B 0,C 180,E1 -9351.591,E2 -9351.591} C_VEL
LIN {X 0,Y 432.594,Z 485.726,A -85,B 0,C 180,E1 -9354.407,E2 -9354.407} C_VEL
LIN {X 0,Y 432.597,Z 485.705,A -85,B 0,C 180,E1 -9358.138,E2 -9358.138} C_VEL
LIN {X 0,Y 432.724,Z 485.698,A -85,B 0,C 180,E1 -9360,E2 -9360} C_VEL
LIN {X 0,Y 432.597,Z 485.72,A -85,B 0,C 180,E1 -9362.794,E2 -9362.794} C_VEL
LIN {X 0,Y 432.564,Z 485.712,A -85,B 0,C 180,E1 -9366.531,E2 -9366.531} C_VEL
LIN {X 0,Y 432.435,Z 485.741,A -85,B 0,C 180,E1 -9369.354,E2 -9369.354} C_VEL
LIN {X 0,Y 432.423,Z 485.729,A -85,B 0,C 180,E1 -9372.804,E2 -9372.804} C_VEL
LIN {X 0,Y 432.405,Z 485.747,A -85,B 0,C 180,E1 -9376.48,E2 -9376.48} C_VEL
LIN {X 0,Y 432.332,Z 485.746,A -85,B 0,C 180,E1 -9379.961,E2 -9379.961} C_VEL
LIN {X 0,Y 432.312,Z 485.759,A -85,B 0,C 180,E1 -9382.965,E2 -9382.965} C_VEL
LIN {X 0,Y 432.358,Z 485.748,A -85,B 0,C 180,E1 -9386.033,E2 -9386.033} C_VEL
LIN {X 0,Y 432.337,Z 485.754,A -85,B 0,C 180,E1 -9389.188,E2 -9389.188} C_VEL
LIN {X 0,Y 432.317,Z 485.752,A -85,B 0,C 180,E1 -9392.444,E2 -9392.444} C_VEL
LIN {X 0,Y 432.341,Z 485.753,A -85,B 0,C 180,E1 -9395.633,E2 -9395.633} C_VEL
LIN {X 0,Y 432.361,Z 485.752,A -85,B 0,C 180,E1 -9399.342,E2 -9399.342} C_VEL
LIN {X 0,Y 432.362,Z 485.746,A -85,B 0,C 180,E1 -9401.794,E2 -9401.794} C_VEL
LIN {X 0,Y 432.33,Z 485.759,A -85,B 0,C 180,E1 -9404.348,E2 -9404.348} C_VEL
LIN {X 0,Y 432.322,Z 485.743,A -85,B 0,C 180,E1 -9407.016,E2 -9407.016} C_VEL
LIN {X 0,Y 432.339,Z 485.754,A -85,B 0,C 180,E1 -9409.82,E2 -9409.82} C_VEL
LIN {X 0,Y 432.304,Z 485.713,A -85,B 0,C 180,E1 -9413.023,E2 -9413.023} C_VEL
LIN {X 0,Y 432.358,Z 485.754,A -85,B 0,C 180,E1 -9415.997,E2 -9415.997} C_VEL
LIN {X 0,Y 432.393,Z 485.772,A -85,B 0,C 180,E1 -9419.11,E2 -9419.11} C_VEL
LIN {X 0,Y 433.386,Z 490.54,A -85,B 0,C 180,E1 -9420.357,E2 -9420.357} C_VEL
LIN {X 0,Y 435.387,Z 500.555,A -85,B 0,C 180,E1 -9422.782,E2 -9422.782} C_VEL
LIN {X 0,Y 435.659,Z 504.476,A -85,B 0,C 180,E1 -9423.665,E2 -9423.665} C_VEL
LIN {X 0,Y 434.72,Z 518.407,A -85,B 0,C 180,E1 -9426.667,E2 -9426.667} C_VEL
LIN {X 0,Y 434.447,Z 522.729,A -85,B 0,C 180,E1 -9427.594,E2 -9427.594} C_VEL
LIN {X 0,Y 435.38,Z 527.545,A -85,B 0,C 180,E1 -9427.775,E2 -9427.775} C_VEL
LIN {X 0,Y 440.119,Z 551.263,A -85,B 0,C 180,E1 -9428.432,E2 -9428.432} C_VEL
LIN {X 0,Y 438.761,Z 656.871,A -85,B 0,C 180,E1 -9430.192,E2 -9430.192} C_VEL
LIN {X 0,Y 438.398,Z 668.27,A -85,B 0,C 180,E1 -9430.48,E2 -9430.48} C_VEL
LIN {X 0,Y 437.912,Z 678.813,A -85,B 0,C 180,E1 -9430.853,E2 -9430.853} C_VEL
LIN {X 0,Y 437.336,Z 690.15,A -85,B 0,C 180,E1 -9431.384,E2 -9431.384} C_VEL
LIN {X 0,Y 436.757,Z 699.737,A -85,B 0,C 180,E1 -9431.941,E2 -9431.941} C_VEL
LIN {X 0,Y 436.053,Z 709.868,A -85,B 0,C 180,E1 -9432.653,E2 -9432.653} C_VEL
LIN {X 0,Y 435.287,Z 719.594,A -85,B 0,C 180,E1 -9433.467,E2 -9433.467} C_VEL
LIN {X 0,Y 434.577,Z 729.018,A -85,B 0,C 180,E1 -9434.404,E2 -9434.404} C_VEL
LIN {X 0,Y 433.805,Z 738.041,A -85,B 0,C 180,E1 -9435.457,E2 -9435.457} C_VEL
LIN {X 0,Y 433.281,Z 745.333,A -85,B 0,C 180,E1 -9436.445,E2 -9436.445} C_VEL
LIN {X 0,Y 432.738,Z 752.631,A -85,B 0,C 180,E1 -9437.589,E2 -9437.589} C_VEL
LIN {X 0,Y 432.219,Z 760.161,A -85,B 0,C 180,E1 -9438.986,E2 -9438.986} C_VEL
LIN {X 0,Y 431.873,Z 765.564,A -85,B 0,C 180,E1 -9440.162,E2 -9440.162} C_VEL
LIN {X 0,Y 431.582,Z 770.996,A -85,B 0,C 180,E1 -9441.573,E2 -9441.573} C_VEL
LIN {X 0,Y 431.41,Z 775.439,A -85,B 0,C 180,E1 -9442.982,E2 -9442.982} C_VEL
LIN {X 0,Y 431.281,Z 778.98,A -85,B 0,C 180,E1 -9444.389,E2 -9444.389} C_VEL
LIN {X 0,Y 431.245,Z 780.918,A -85,B 0,C 180,E1 -9445.326,E2 -9445.326} C_VEL
LIN {X 0,Y 431.231,Z 783.598,A -85,B 0,C 180,E1 -9447.198,E2 -9447.198} C_VEL
LIN {X 0,Y 431.167,Z 784.883,A -85,B 0,C 180,E1 -9449.066,E2 -9449.066} C_VEL
LIN {X 0,Y 431.166,Z 785.134,A -85,B 0,C 180,E1 -9450,E2 -9450} C_VEL
LIN {X 0,Y 431.2,Z 784.412,A -85,B 0,C 180,E1 -9451.868,E2 -9451.868} C_VEL
LIN {X 0,Y 431.231,Z 783.598,A -85,B 0,C 180,E1 -9452.802,E2 -9452.802} C_VEL
LIN {X 0,Y 431.245,Z 780.918,A -85,B 0,C 180,E1 -9454.674,E2 -9454.674} C_VEL
LIN {X 0,Y 431.373,Z 776.705,A -85,B 0,C 180,E1 -9456.548,E2 -9456.548} C_VEL
LIN {X 0,Y 431.485,Z 772.574,A -85,B 0,C 180,E1 -9457.958,E2 -9457.958} C_VEL
LIN {X 0,Y 431.75,Z 767.477,A -85,B 0,C 180,E1 -9459.368,E2 -9459.368} C_VEL
LIN {X 0,Y 432.111,Z 761.298,A -85,B 0,C 180,E1 -9460.78,E2 -9460.78} C_VEL
LIN {X 0,Y 432.584,Z 755.224,A -85,B 0,C 180,E1 -9461.955,E2 -9461.955} C_VEL
LIN {X 0,Y 433.008,Z 748.144,A -85,B 0,C 180,E1 -9463.134,E2 -9463.134} C_VEL
LIN {X 0,Y 433.528,Z 741.681,A -85,B 0,C 180,E1 -9464.073,E2 -9464.073} C_VEL
LIN {X 0,Y 434.262,Z 732.196,A -85,B 0,C 180,E1 -9465.247,E2 -9465.247} C_VEL
LIN {X 0,Y 434.968,Z 723.316,A -85,B 0,C 180,E1 -9466.183,E2 -9466.183} C_VEL
LIN {X 0,Y 435.758,Z 714.263,A -85,B 0,C 180,E1 -9466.997,E2 -9466.997} C_VEL
LIN {X 0,Y 436.506,Z 703.453,A -85,B 0,C 180,E1 -9467.813,E2 -9467.813} C_VEL
LIN {X 0,Y 437.168,Z 692.884,A -85,B 0,C 180,E1 -9468.468,E2 -9468.468} C_VEL
LIN {X 0,Y 437.746,Z 681.533,A -85,B 0,C 180,E1 -9469.033,E2 -9469.033} C_VEL
LIN {X 0,Y 438.308,Z 671.007,A -85,B 0,C 180,E1 -9469.433,E2 -9469.433} C_VEL
LIN {X 0,Y 438.699,Z 659.591,A -85,B 0,C 180,E1 -9469.75,E2 -9469.75} C_VEL
LIN {X 0,Y 439.24,Z 629.48,A -85,B 0,C 180,E1 -9470.273,E2 -9470.273} C_VEL
LIN {X 0,Y 440.02,Z 550.581,A -85,B 0,C 180,E1 -9471.585,E2 -9471.585} C_VEL
LIN {X 0,Y 434.497,Z 523.081,A -85,B 0,C 180,E1 -9472.369,E2 -9472.369} C_VEL
LIN {X 0,Y 434.496,Z 521.721,A -85,B 0,C 180,E1 -9472.591,E2 -9472.591} C_VEL
LIN {X 0,Y 435.591,Z 507.008,A -85,B 0,C 180,E1 -9475.825,E2 -9475.825} C_VEL
LIN {X 0,Y 435.707,Z 502.373,A -85,B 0,C 180,E1 -9476.848,E2 -9476.848} C_VEL
LIN {X 0,Y 433.642,Z 491.704,A -85,B 0,C 180,E1 -9479.357,E2 -9479.357} C_VEL
LIN {X 0,Y 432.441,Z 486.039,A -85,B 0,C 180,E1 -9480.775,E2 -9480.775} C_VEL
LIN {X 0,Y 432.367,Z 485.72,A -85,B 0,C 180,E1 -9481.004,E2 -9481.004} C_VEL
LIN {X 0,Y 432.338,Z 485.737,A -85,B 0,C 180,E1 -9484.676,E2 -9484.676} C_VEL
LIN {X 0,Y 432.337,Z 485.728,A -85,B 0,C 180,E1 -9488.149,E2 -9488.149} C_VEL
LIN {X 0,Y 432.331,Z 485.751,A -85,B 0,C 180,E1 -9491.601,E2 -9491.601} C_VEL
LIN {X 0,Y 432.337,Z 485.745,A -85,B 0,C 180,E1 -9494.346,E2 -9494.346} C_VEL
LIN {X 0,Y 432.316,Z 485.76,A -85,B 0,C 180,E1 -9497.015,E2 -9497.015} C_VEL
LIN {X 0,Y 432.351,Z 485.753,A -85,B 0,C 180,E1 -9499.816,E2 -9499.816} C_VEL
LIN {X 0,Y 432.311,Z 485.754,A -85,B 0,C 180,E1 -9503.022,E2 -9503.022} C_VEL
LIN {X 0,Y 432.354,Z 485.745,A -85,B 0,C 180,E1 -9505.996,E2 -9505.996} C_VEL
LIN {X 0,Y 432.341,Z 485.758,A -85,B 0,C 180,E1 -9509.489,E2 -9509.489} C_VEL
LIN {X 0,Y 432.387,Z 485.737,A -85,B 0,C 180,E1 -9512.928,E2 -9512.928} C_VEL
LIN {X 0,Y 432.364,Z 485.75,A -85,B 0,C 180,E1 -9516.023,E2 -9516.023} C_VEL
LIN {X 0,Y 432.343,Z 485.743,A -85,B 0,C 180,E1 -9519.045,E2 -9519.045} C_VEL
LIN {X 0,Y 432.371,Z 485.749,A -85,B 0,C 180,E1 -9522.01,E2 -9522.01} C_VEL
LIN {X 0,Y 432.387,Z 485.745,A -85,B 0,C 180,E1 -9524.926,E2 -9524.926} C_VEL
LIN {X 0,Y 432.451,Z 485.735,A -85,B 0,C 180,E1 -9527.803,E2 -9527.803} C_VEL
LIN {X 0,Y 432.484,Z 485.735,A -85,B 0,C 180,E1 -9531.59,E2 -9531.59} C_VEL
LIN {X 0,Y 432.589,Z 485.703,A -85,B 0,C 180,E1 -9534.406,E2 -9534.406} C_VEL
LIN {X 0,Y 432.597,Z 485.72,A -85,B 0,C 180,E1 -9538.138,E2 -9538.138} C_VEL
LIN {X 0,Y 432.724,Z 485.698,A -85,B 0,C 180,E1 -9540,E2 -9540} C_VEL
LIN {X 0,Y 432.597,Z 485.704,A -85,B 0,C 180,E1 -9542.793,E2 -9542.793} C_VEL
LIN {X 0,Y 432.563,Z 485.723,A -85,B 0,C 180,E1 -9546.53,E2 -9546.53} C_VEL
LIN {X 0,Y 432.434,Z 485.73,A -85,B 0,C 180,E1 -9549.353,E2 -9549.353} C_VEL
LIN {X 0,Y 432.421,Z 485.741,A -85,B 0,C 180,E1 -9552.803,E2 -9552.803} C_VEL
LIN {X 0,Y 432.403,Z 485.734,A -85,B 0,C 180,E1 -9556.479,E2 -9556.479} C_VEL
LIN {X 0,Y 432.33,Z 485.757,A -85,B 0,C 180,E1 -9559.96,E2 -9559.96} C_VEL
LIN {X 0,Y 432.309,Z 485.753,A -85,B 0,C 180,E1 -9562.964,E2 -9562.964} C_VEL
LIN {X 0,Y 432.356,Z 485.753,A -85,B 0,C 180,E1 -9566.032,E2 -9566.032} C_VEL
LIN {X 0,Y 432.343,Z 485.752,A -85,B 0,C 180,E1 -9569.187,E2 -9569.187} C_VEL
LIN {X 0,Y 432.323,Z 485.755,A -85,B 0,C 180,E1 -9572.295,E2 -9572.295} C_VEL
LIN {X 0,Y 432.332,Z 485.751,A -85,B 0,C 180,E1 -9574.677,E2 -9574.677} C_VEL
LIN {X 0,Y 432.339,Z 485.756,A -85,B 0,C 180,E1 -9578.149,E2 -9578.149} C_VEL
LIN {X 0,Y 432.362,Z 485.75,A -85,B 0,C 180,E1 -9581.793,E2 -9581.793} C_VEL
LIN {X 0,Y 432.371,Z 485.745,A -85,B 0,C 180,E1 -9584.342,E2 -9584.342} C_VEL
LIN {X 0,Y 432.358,Z 485.721,A -85,B 0,C 180,E1 -9587.009,E2 -9587.009} C_VEL
LIN {X 0,Y 432.354,Z 485.755,A -85,B 0,C 180,E1 -9589.817,E2 -9589.817} C_VEL
LIN {X 0,Y 432.31,Z 485.741,A -85,B 0,C 180,E1 -9593.023,E2 -9593.023} C_VEL
LIN {X 0,Y 432.353,Z 485.757,A -85,B 0,C 180,E1 -9595.997,E2 -9595.997} C_VEL
LIN {X 0,Y 432.389,Z 485.753,A -85,B 0,C 180,E1 -9599.744,E2 -9599.744} C_VEL
LIN {X 0,Y 432.394,Z 485.751,A -85,B 0,C 180,E1 -9603.373,E2 -9603.373} C_VEL
LIN {X 0,Y 432.366,Z 485.755,A -85,B 0,C 180,E1 -9606.024,E2 -9606.024} C_VEL
LIN {X 0,Y 432.345,Z 485.755,A -85,B 0,C 180,E1 -9609.046,E2 -9609.046} C_VEL
LIN {X 0,Y 432.374,Z 485.755,A -85,B 0,C 180,E1 -9612.011,E2 -9612.011} C_VEL
LIN {X 0,Y 432.391,Z 485.75,A -85,B 0,C 180,E1 -9614.927,E2 -9614.927} C_VEL
LIN {X 0,Y 432.455,Z 485.744,A -85,B 0,C 180,E1 -9617.804,E2 -9617.804} C_VEL
LIN {X 0,Y 432.488,Z 485.74,A -85,B 0,C 180,E1 -9621.59,E2 -9621.59} C_VEL
LIN {X 0,Y 432.594,Z 485.726,A -85,B 0,C 180,E1 -9624.406,E2 -9624.406} C_VEL
LIN {X 0,Y 432.602,Z 485.726,A -85,B 0,C 180,E1 -9628.138,E2 -9628.138} C_VEL
LIN {X 0,Y 432.73,Z 485.711,A -85,B 0,C 180,E1 -9630,E2 -9630} C_VEL
LIN {X 0,Y 432.602,Z 485.725,A -85,B 0,C 180,E1 -9632.794,E2 -9632.794} C_VEL
LIN {X 0,Y 432.463,Z 485.741,A -85,B 0,C 180,E1 -9635.041,E2 -9635.041} C_VEL
LIN {X 0,Y 431.904,Z 485.813,A -85,B 0,C 180,E1 -9635.82,E2 -9635.82} C_VEL
LIN {X 0,Y 429.056,Z 486.166,A -85,B 0,C 180,E1 -9637.085,E2 -9637.085} C_VEL
LIN {X 0,Y 426.57,Z 486.477,A -85,B 0,C 180,E1 -9638.106,E2 -9638.106} C_VEL
LIN {X 0,Y 425.489,Z 486.61,A -85,B 0,C 180,E1 -9638.895,E2 -9638.895} C_VEL
LIN {X 0,Y 425.398,Z 486.621,A -85,B 0,C 180,E1 -9639.163,E2 -9639.163} C_VEL
LIN {X 0,Y 425.389,Z 486.623,A -85,B 0,C 180,E1 -9642.904,E2 -9642.904} C_VEL
LIN {X 0,Y 425.357,Z 486.627,A -85,B 0,C 180,E1 -9646.605,E2 -9646.605} C_VEL
LIN {X 0,Y 425.324,Z 486.631,A -85,B 0,C 180,E1 -9649.635,E2 -9649.635} C_VEL
LIN {X 0,Y 425.302,Z 486.633,A -85,B 0,C 180,E1 -9653.365,E2 -9653.365} C_VEL
LIN {X 0,Y 425.343,Z 486.628,A -85,B 0,C 180,E1 -9656.844,E2 -9656.844} C_VEL
LIN {X 0,Y 425.313,Z 486.632,A -85,B 0,C 180,E1 -9659.717,E2 -9659.717} C_VEL
LIN {X 0,Y 425.276,Z 486.635,A -85,B 0,C 180,E1 -9663.048,E2 -9663.048} C_VEL
LIN {X 0,Y 425.278,Z 486.62,A -85,B 0,C 180,E1 -9665.929,E2 -9665.929} C_VEL
LIN {X 0,Y 425.307,Z 486.63,A -85,B 0,C 180,E1 -9669.046,E2 -9669.046} C_VEL
LIN {X 0,Y 425.324,Z 486.598,A -85,B 0,C 180,E1 -9672.646,E2 -9672.646} C_VEL
LIN {X 0,Y 425.327,Z 486.626,A -85,B 0,C 180,E1 -9676.053,E2 -9676.053} C_VEL
LIN {X 0,Y 425.294,Z 486.625,A -85,B 0,C 180,E1 -9678.625,E2 -9678.625} C_VEL
LIN {X 0,Y 425.307,Z 486.63,A -85,B 0,C 180,E1 -9681.103,E2 -9681.103} C_VEL
LIN {X 0,Y 425.292,Z 486.629,A -85,B 0,C 180,E1 -9684.664,E2 -9684.664} C_VEL
LIN {X 0,Y 425.264,Z 486.635,A -85,B 0,C 180,E1 -9688.074,E2 -9688.074} C_VEL
LIN {X 0,Y 425.329,Z 486.624,A -85,B 0,C 180,E1 -9691.368,E2 -9691.368} C_VEL
LIN {X 0,Y 425.286,Z 486.624,A -85,B 0,C 180,E1 -9694.555,E2 -9694.555} C_VEL
LIN {X 0,Y 425.278,Z 486.629,A -85,B 0,C 180,E1 -9697.661,E2 -9697.661} C_VEL
LIN {X 0,Y 425.352,Z 486.619,A -85,B 0,C 180,E1 -9700.704,E2 -9700.704} C_VEL
LIN {X 0,Y 425.379,Z 486.609,A -85,B 0,C 180,E1 -9703.688,E2 -9703.688} C_VEL
LIN {X 0,Y 425.403,Z 486.615,A -85,B 0,C 180,E1 -9707.598,E2 -9707.598} C_VEL
LIN {X 0,Y 425.433,Z 486.603,A -85,B 0,C 180,E1 -9711.45,E2 -9711.45} C_VEL
LIN {X 0,Y 425.569,Z 486.6,A -85,B 0,C 180,E1 -9714.314,E2 -9714.314} C_VEL
LIN {X 0,Y 425.566,Z 486.579,A -85,B 0,C 180,E1 -9718.108,E2 -9718.108} C_VEL
LIN {X 0,Y 425.694,Z 486.574,A -85,B 0,C 180,E1 -9720,E2 -9720} C_VEL
LIN {X 0,Y 425.549,Z 486.597,A -85,B 0,C 180,E1 -9722.84,E2 -9722.84} C_VEL
LIN {X 0,Y 425.522,Z 486.59,A -85,B 0,C 180,E1 -9726.639,E2 -9726.639} C_VEL
LIN {X 0,Y 425.393,Z 486.618,A -85,B 0,C 180,E1 -9729.51,E2 -9729.51} C_VEL
LIN {X 0,Y 425.385,Z 486.604,A -85,B 0,C 180,E1 -9732.904,E2 -9732.904} C_VEL
LIN {X 0,Y 425.354,Z 486.628,A -85,B 0,C 180,E1 -9736.606,E2 -9736.606} C_VEL
LIN {X 0,Y 425.321,Z 486.618,A -85,B 0,C 180,E1 -9739.636,E2 -9739.636} C_VEL
LIN {X 0,Y 425.281,Z 486.627,A -85,B 0,C 180,E1 -9742.339,E2 -9742.339} C_VEL
LIN {X 0,Y 425.289,Z 486.627,A -85,B 0,C 180,E1 -9745.446,E2 -9745.446} C_VEL
LIN {X 0,Y 425.325,Z 486.624,A -85,B 0,C 180,E1 -9748.633,E2 -9748.633} C_VEL
LIN {X 0,Y 425.259,Z 486.632,A -85,B 0,C 180,E1 -9751.928,E2 -9751.928} C_VEL
LIN {X 0,Y 425.295,Z 486.632,A -85,B 0,C 180,E1 -9755.337,E2 -9755.337} C_VEL
LIN {X 0,Y 425.307,Z 486.633,A -85,B 0,C 180,E1 -9759.047,E2 -9759.047} C_VEL
LIN {X 0,Y 425.311,Z 486.625,A -85,B 0,C 180,E1 -9761.963,E2 -9761.963} C_VEL
LIN {X 0,Y 425.286,Z 486.626,A -85,B 0,C 180,E1 -9765.283,E2 -9765.283} C_VEL
LIN {X 0,Y 425.274,Z 486.633,A -85,B 0,C 180,E1 -9768.623,E2 -9768.623} C_VEL
LIN {X 0,Y 425.31,Z 486.615,A -85,B 0,C 180,E1 -9771.104,E2 -9771.104} C_VEL
LIN {X 0,Y 425.297,Z 486.595,A -85,B 0,C 180,E1 -9774.665,E2 -9774.665} C_VEL
LIN {X 0,Y 425.274,Z 486.61,A -85,B 0,C 180,E1 -9778.075,E2 -9778.075} C_VEL
LIN {X 0,Y 425.344,Z 486.732,A -85,B 0,C 180,E1 -9778.845,E2 -9778.845} C_VEL
LIN {X 0,Y 427.803,Z 498.288,A -85,B 0,C 180,E1 -9781.792,E2 -9781.792} C_VEL
LIN {X 0,Y 428.791,Z 504.28,A -85,B 0,C 180,E1 -9783.21,E2 -9783.21} C_VEL
LIN {X 0,Y 427.966,Z 517.087,A -85,B 0,C 180,E1 -9786.019,E2 -9786.019} C_VEL
LIN {X 0,Y 427.567,Z 522.536,A -85,B 0,C 180,E1 -9787.216,E2 -9787.216} C_VEL
LIN {X 0,Y 428.634,Z 527.975,A -85,B 0,C 180,E1 -9787.417,E2 -9787.417} C_VEL
LIN {X 0,Y 433.513,Z 552.295,A -85,B 0,C 180,E1 -9788.108,E2 -9788.108} C_VEL
LIN {X 0,Y 432.099,Z 656.674,A -85,B 0,C 180,E1 -9789.874,E2 -9789.874} C_VEL
LIN {X 0,Y 431.721,Z 668.072,A -85,B 0,C 180,E1 -9790.165,E2 -9790.165} C_VEL
LIN {X 0,Y 431.208,Z 678.615,A -85,B 0,C 180,E1 -9790.544,E2 -9790.544} C_VEL
LIN {X 0,Y 430.672,Z 688.956,A -85,B 0,C 180,E1 -9791.028,E2 -9791.028} C_VEL
LIN {X 0,Y 429.959,Z 700.035,A -85,B 0,C 180,E1 -9791.681,E2 -9791.681} C_VEL
LIN {X 0,Y 429.269,Z 709.669,A -85,B 0,C 180,E1 -9792.37,E2 -9792.37} C_VEL
LIN {X 0,Y 428.467,Z 719.396,A -85,B 0,C 180,E1 -9793.197,E2 -9793.197} C_VEL
LIN {X 0,Y 427.668,Z 728.818,A -85,B 0,C 180,E1 -9794.145,E2 -9794.145} C_VEL
LIN {X 0,Y 426.87,Z 737.841,A -85,B 0,C 180,E1 -9795.215,E2 -9795.215} C_VEL
LIN {X 0,Y 426.329,Z 744.82,A -85,B 0,C 180,E1 -9796.171,E2 -9796.171} C_VEL
LIN {X 0,Y 425.747,Z 752.591,A -85,B 0,C 180,E1 -9797.41,E2 -9797.41} C_VEL
LIN {X 0,Y 425.211,Z 759.962,A -85,B 0,C 180,E1 -9798.802,E2 -9798.802} C_VEL
LIN {X 0,Y 424.817,Z 765.364,A -85,B 0,C 180,E1 -9799.997,E2 -9799.997} C_VEL
LIN {X 0,Y 424.506,Z 770.796,A -85,B 0,C 180,E1 -9801.431,E2 -9801.431} C_VEL
LIN {X 0,Y 424.328,Z 775.24,A -85,B 0,C 180,E1 -9802.864,E2 -9802.864} C_VEL
LIN {X 0,Y 424.195,Z 778.781,A -85,B 0,C 180,E1 -9804.295,E2 -9804.295} C_VEL
LIN {X 0,Y 424.172,Z 780.72,A -85,B 0,C 180,E1 -9805.248,E2 -9805.248} C_VEL
LIN {X 0,Y 424.127,Z 783.399,A -85,B 0,C 180,E1 -9807.151,E2 -9807.151} C_VEL
LIN {X 0,Y 424.086,Z 784.685,A -85,B 0,C 180,E1 -9809.05,E2 -9809.05} C_VEL
LIN {X 0,Y 424.083,Z 784.937,A -85,B 0,C 180,E1 -9810,E2 -9810} C_VEL
LIN {X 0,Y 424.126,Z 784.215,A -85,B 0,C 180,E1 -9811.899,E2 -9811.899} C_VEL
LIN {X 0,Y 424.127,Z 783.399,A -85,B 0,C 180,E1 -9812.849,E2 -9812.849} C_VEL
LIN {X 0,Y 424.171,Z 780.72,A -85,B 0,C 180,E1 -9814.752,E2 -9814.752} C_VEL
LIN {X 0,Y 424.296,Z 776.506,A -85,B 0,C 180,E1 -9816.658,E2 -9816.658} C_VEL
LIN {X 0,Y 424.42,Z 772.375,A -85,B 0,C 180,E1 -9818.091,E2 -9818.091} C_VEL
LIN {X 0,Y 424.706,Z 767.277,A -85,B 0,C 180,E1 -9819.525,E2 -9819.525} C_VEL
LIN {X 0,Y 425.102,Z 761.099,A -85,B 0,C 180,E1 -9820.96,E2 -9820.96} C_VEL
LIN {X 0,Y 425.574,Z 755.024,A -85,B 0,C 180,E1 -9822.155,E2 -9822.155} C_VEL
LIN {X 0,Y 426.05,Z 747.945,A -85,B 0,C 180,E1 -9823.352,E2 -9823.352} C_VEL
LIN {X 0,Y 426.743,Z 739.662,A -85,B 0,C 180,E1 -9824.545,E2 -9824.545} C_VEL
LIN {X 0,Y 427.469,Z 730.937,A -85,B 0,C 180,E1 -9825.618,E2 -9825.618} C_VEL
LIN {X 0,Y 428.25,Z 721.877,A -85,B 0,C 180,E1 -9826.567,E2 -9826.567} C_VEL
LIN {X 0,Y 429.017,Z 712.598,A -85,B 0,C 180,E1 -9827.395,E2 -9827.395} C_VEL
LIN {X 0,Y 429.729,Z 703.254,A -85,B 0,C 180,E1 -9828.103,E2 -9828.103} C_VEL
LIN {X 0,Y 430.356,Z 693.841,A -85,B 0,C 180,E1 -9828.705,E2 -9828.705} C_VEL
LIN {X 0,Y 430.958,Z 682.695,A -85,B 0,C 180,E1 -9829.283,E2 -9829.283} C_VEL
LIN {X 0,Y 431.625,Z 670.809,A -85,B 0,C 180,E1 -9829.746,E2 -9829.746} C_VEL
LIN {X 0,Y 432.039,Z 659.393,A -85,B 0,C 180,E1 -9830.067,E2 -9830.067} C_VEL
LIN {X 0,Y 432.582,Z 629.282,A -85,B 0,C 180,E1 -9830.599,E2 -9830.599} C_VEL
LIN {X 0,Y 433.538,Z 552.296,A -85,B 0,C 180,E1 -9831.891,E2 -9831.891} C_VEL
LIN {X 0,Y 427.611,Z 522.797,A -85,B 0,C 180,E1 -9832.755,E2 -9832.755} C_VEL
LIN {X 0,Y 427.731,Z 520.419,A -85,B 0,C 180,E1 -9833.224,E2 -9833.224} C_VEL
LIN {X 0,Y 428.82,Z 505.661,A -85,B 0,C 180,E1 -9836.525,E2 -9836.525} C_VEL
LIN {X 0,Y 428.334,Z 500.971,A -85,B 0,C 180,E1 -9837.622,E2 -9837.622} C_VEL
LIN {X 0,Y 425.87,Z 489.195,A -85,B 0,C 180,E1 -9840.494,E2 -9840.494} C_VEL
LIN {X 0,Y 425.312,Z 486.638,A -85,B 0,C 180,E1 -9841.227,E2 -9841.227} C_VEL
LIN {X 0,Y 425.31,Z 486.621,A -85,B 0,C 180,E1 -9844.287,E2 -9844.287} C_VEL
LIN {X 0,Y 425.278,Z 486.595,A -85,B 0,C 180,E1 -9847.693,E2 -9847.693} C_VEL
LIN {X 0,Y 425.282,Z 486.634,A -85,B 0,C 180,E1 -9850.52,E2 -9850.52} C_VEL
LIN {X 0,Y 425.265,Z 486.623,A -85,B 0,C 180,E1 -9853.954,E2 -9853.954} C_VEL
LIN {X 0,Y 425.278,Z 486.632,A -85,B 0,C 180,E1 -9857.347,E2 -9857.347} C_VEL
LIN {X 0,Y 425.304,Z 486.631,A -85,B 0,C 180,E1 -9859.874,E2 -9859.874} C_VEL
LIN {X 0,Y 425.281,Z 486.626,A -85,B 0,C 180,E1 -9862.486,E2 -9862.486} C_VEL
LIN {X 0,Y 425.303,Z 486.624,A -85,B 0,C 180,E1 -9865.816,E2 -9865.816} C_VEL
LIN {X 0,Y 425.285,Z 486.635,A -85,B 0,C 180,E1 -9869.238,E2 -9869.238} C_VEL
LIN {X 0,Y 425.344,Z 486.614,A -85,B 0,C 180,E1 -9872.442,E2 -9872.442} C_VEL
LIN {X 0,Y 425.345,Z 486.628,A -85,B 0,C 180,E1 -9875.601,E2 -9875.601} C_VEL
LIN {X 0,Y 425.286,Z 486.623,A -85,B 0,C 180,E1 -9878.681,E2 -9878.681} C_VEL
LIN {X 0,Y 425.326,Z 486.63,A -85,B 0,C 180,E1 -9881.702,E2 -9881.702} C_VEL
LIN {X 0,Y 425.34,Z 486.621,A -85,B 0,C 180,E1 -9884.67,E2 -9884.67} C_VEL
LIN {X 0,Y 425.404,Z 486.608,A -85,B 0,C 180,E1 -9887.598,E2 -9887.598} C_VEL
LIN {X 0,Y 425.434,Z 486.615,A -85,B 0,C 180,E1 -9891.449,E2 -9891.449} C_VEL
LIN {X 0,Y 425.546,Z 486.58,A -85,B 0,C 180,E1 -9894.313,E2 -9894.313} C_VEL
LIN {X 0,Y 425.567,Z 486.596,A -85,B 0,C 180,E1 -9898.107,E2 -9898.107} C_VEL
LIN {X 0,Y 425.694,Z 486.574,A -85,B 0,C 180,E1 -9900,E2 -9900} C_VEL
LIN {X 0,Y 425.549,Z 486.582,A -85,B 0,C 180,E1 -9902.839,E2 -9902.839} C_VEL
LIN {X 0,Y 425.52,Z 486.6,A -85,B 0,C 180,E1 -9906.65,E2 -9906.65} C_VEL
LIN {X 0,Y 425.392,Z 486.605,A -85,B 0,C 180,E1 -9909.509,E2 -9909.509} C_VEL
LIN {X 0,Y 425.384,Z 486.618,A -85,B 0,C 180,E1 -9912.903,E2 -9912.903} C_VEL
LIN {X 0,Y 425.352,Z 486.612,A -85,B 0,C 180,E1 -9916.605,E2 -9916.605} C_VEL
LIN {X 0,Y 425.319,Z 486.628,A -85,B 0,C 180,E1 -9919.636,E2 -9919.636} C_VEL
LIN {X 0,Y 425.297,Z 486.625,A -85,B 0,C 180,E1 -9923.365,E2 -9923.365} C_VEL
LIN {X 0,Y 425.34,Z 486.624,A -85,B 0,C 180,E1 -9926.845,E2 -9926.845} C_VEL
LIN {X 0,Y 425.309,Z 486.622,A -85,B 0,C 180,E1 -9929.717,E2 -9929.717} C_VEL
LIN {X 0,Y 425.275,Z 486.633,A -85,B 0,C 180,E1 -9933.048,E2 -9933.048} C_VEL
LIN {X 0,Y 425.276,Z 486.627,A -85,B 0,C 180,E1 -9935.929,E2 -9935.929} C_VEL
LIN {X 0,Y 425.295,Z 486.632,A -85,B 0,C 180,E1 -9939.045,E2 -9939.045} C_VEL
LIN {X 0,Y 425.323,Z 486.628,A -85,B 0,C 180,E1 -9942.646,E2 -9942.646} C_VEL
LIN {X 0,Y 425.311,Z 486.603,A -85,B 0,C 180,E1 -9946.052,E2 -9946.052} C_VEL
LIN {X 0,Y 425.303,Z 486.625,A -85,B 0,C 180,E1 -9948.626,E2 -9948.626} C_VEL
LIN {X 0,Y 425.319,Z 486.629,A -85,B 0,C 180,E1 -9951.105,E2 -9951.105} C_VEL
LIN {X 0,Y 425.294,Z 486.629,A -85,B 0,C 180,E1 -9954.665,E2 -9954.665} C_VEL
LIN {X 0,Y 425.261,Z 486.64,A -85,B 0,C 180,E1 -9958.074,E2 -9958.074} C_VEL
LIN {X 0,Y 425.332,Z 486.63,A -85,B 0,C 180,E1 -9961.369,E2 -9961.369} C_VEL
LIN {X 0,Y 425.29,Z 486.635,A -85,B 0,C 180,E1 -9964.555,E2 -9964.555} C_VEL
LIN {X 0,Y 425.283,Z 486.638,A -85,B 0,C 180,E1 -9967.662,E2 -9967.662} C_VEL
LIN {X 0,Y 425.357,Z 486.626,A -85,B 0,C 180,E1 -9970.704,E2 -9970.704} C_VEL
LIN {X 0,Y 425.384,Z 486.625,A -85,B 0,C 180,E1 -9973.688,E2 -9973.688} C_VEL
LIN {X 0,Y 425.408,Z 486.622,A -85,B 0,C 180,E1 -9977.598,E2 -9977.598} C_VEL
LIN {X 0,Y 425.439,Z 486.618,A -85,B 0,C 180,E1 -9981.45,E2 -9981.45} C_VEL
LIN {X 0,Y 425.55,Z 486.604,A -85,B 0,C 180,E1 -9984.313,E2 -9984.313} C_VEL
LIN {X 0,Y 425.572,Z 486.602,A -85,B 0,C 180,E1 -9988.107,E2 -9988.107} C_VEL
LIN {X 0,Y 425.7,Z 486.586,A -85,B 0,C 180,E1 -9990,E2 -9990} C_VEL
LIN {X 0,Y 425.553,Z 486.603,A -85,B 0,C 180,E1 -9992.84,E2 -9992.84} C_VEL
LIN {X 0,Y 425.527,Z 486.607,A -85,B 0,C 180,E1 -9996.639,E2 -9996.639} C_VEL
LIN {X 0,Y 425.398,Z 486.621,A -85,B 0,C 180,E1 -9999.163,E2 -9999.163} C_VEL
LIN {X 0,Y 424.727,Z 486.707,A -85,B 0,C 180,E1 -9999.953,E2 -9999.953} C_VEL
LIN {X 0,Y 421.878,Z 487.06,A -85,B 0,C 180,E1 -10001.237,E2 -10001.237} C_VEL
LIN {X 0,Y 419.461,Z 487.363,A -85,B 0,C 180,E1 -10002.273,E2 -10002.273} C_VEL
LIN {X 0,Y 418.411,Z 487.492,A -85,B 0,C 180,E1 -10003.073,E2 -10003.073} C_VEL
LIN {X 0,Y 418.318,Z 487.503,A -85,B 0,C 180,E1 -10003.345,E2 -10003.345} C_VEL
LIN {X 0,Y 418.308,Z 487.506,A -85,B 0,C 180,E1 -10006.735,E2 -10006.735} C_VEL
LIN {X 0,Y 418.266,Z 487.511,A -85,B 0,C 180,E1 -10009.79,E2 -10009.79} C_VEL
LIN {X 0,Y 418.233,Z 487.514,A -85,B 0,C 180,E1 -10012.736,E2 -10012.736} C_VEL
LIN {X 0,Y 418.266,Z 487.511,A -85,B 0,C 180,E1 -10015.904,E2 -10015.904} C_VEL
LIN {X 0,Y 418.269,Z 487.508,A -85,B 0,C 180,E1 -10019.161,E2 -10019.161} C_VEL
LIN {X 0,Y 418.251,Z 487.511,A -85,B 0,C 180,E1 -10022.844,E2 -10022.844} C_VEL
LIN {X 0,Y 418.242,Z 487.493,A -85,B 0,C 180,E1 -10026.238,E2 -10026.238} C_VEL
LIN {X 0,Y 418.26,Z 487.51,A -85,B 0,C 180,E1 -10029.68,E2 -10029.68} C_VEL
LIN {X 0,Y 418.277,Z 487.478,A -85,B 0,C 180,E1 -10032.329,E2 -10032.329} C_VEL
LIN {X 0,Y 418.267,Z 487.501,A -85,B 0,C 180,E1 -10035.114,E2 -10035.114} C_VEL
LIN {X 0,Y 418.283,Z 487.507,A -85,B 0,C 180,E1 -10037.773,E2 -10037.773} C_VEL
LIN {X 0,Y 418.252,Z 487.509,A -85,B 0,C 180,E1 -10041.559,E2 -10041.559} C_VEL
LIN {X 0,Y 418.251,Z 487.505,A -85,B 0,C 180,E1 -10045.159,E2 -10045.159} C_VEL
LIN {X 0,Y 418.24,Z 487.509,A -85,B 0,C 180,E1 -10047.472,E2 -10047.472} C_VEL
LIN {X 0,Y 418.268,Z 487.505,A -85,B 0,C 180,E1 -10050.893,E2 -10050.893} C_VEL
LIN {X 0,Y 418.262,Z 487.506,A -85,B 0,C 180,E1 -10054.096,E2 -10054.096} C_VEL
LIN {X 0,Y 418.229,Z 487.506,A -85,B 0,C 180,E1 -10057.264,E2 -10057.264} C_VEL
LIN {X 0,Y 418.274,Z 487.505,A -85,B 0,C 180,E1 -10060.364,E2 -10060.364} C_VEL
LIN {X 0,Y 418.307,Z 487.489,A -85,B 0,C 180,E1 -10063.405,E2 -10063.405} C_VEL
LIN {X 0,Y 418.337,Z 487.497,A -85,B 0,C 180,E1 -10067,E2 -10067} C_VEL
LIN {X 0,Y 418.333,Z 487.483,A -85,B 0,C 180,E1 -10070.329,E2 -10070.329} C_VEL
LIN {X 0,Y 418.486,Z 487.477,A -85,B 0,C 180,E1 -10073.249,E2 -10073.249} C_VEL
LIN {X 0,Y 418.337,Z 487.493,A -85,B 0,C 180,E1 -10075.182,E2 -10075.182} C_VEL
LIN {X 0,Y 418.536,Z 487.454,A -85,B 0,C 180,E1 -10078.076,E2 -10078.076} C_VEL
LIN {X 0,Y 418.663,Z 487.449,A -85,B 0,C 180,E1 -10080,E2 -10080} C_VEL
LIN {X 0,Y 418.503,Z 487.474,A -85,B 0,C 180,E1 -10082.888,E2 -10082.888} C_VEL
LIN {X 0,Y 418.485,Z 487.468,A -85,B 0,C 180,E1 -10086.752,E2 -10086.752} C_VEL
LIN {X 0,Y 418.333,Z 487.498,A -85,B 0,C 180,E1 -10089.672,E2 -10089.672} C_VEL
LIN {X 0,Y 418.338,Z 487.48,A -85,B 0,C 180,E1 -10093.001,E2 -10093.001} C_VEL
LIN {X 0,Y 418.305,Z 487.506,A -85,B 0,C 180,E1 -10096.736,E2 -10096.736} C_VEL
LIN {X 0,Y 418.264,Z 487.497,A -85,B 0,C 180,E1 -10099.791,E2 -10099.791} C_VEL
LIN {X 0,Y 418.225,Z 487.512,A -85,B 0,C 180,E1 -10102.737,E2 -10102.737} C_VEL
LIN {X 0,Y 418.265,Z 487.503,A -85,B 0,C 180,E1 -10105.905,E2 -10105.905} C_VEL
LIN {X 0,Y 418.259,Z 487.508,A -85,B 0,C 180,E1 -10109.163,E2 -10109.163} C_VEL
LIN {X 0,Y 418.252,Z 487.5,A -85,B 0,C 180,E1 -10112.845,E2 -10112.845} C_VEL
LIN {X 0,Y 418.244,Z 487.511,A -85,B 0,C 180,E1 -10116.239,E2 -10116.239} C_VEL
LIN {X 0,Y 418.261,Z 487.508,A -85,B 0,C 180,E1 -10119.681,E2 -10119.681} C_VEL
LIN {X 0,Y 418.241,Z 487.507,A -85,B 0,C 180,E1 -10122.324,E2 -10122.324} C_VEL
LIN {X 0,Y 418.236,Z 487.505,A -85,B 0,C 180,E1 -10125.11,E2 -10125.11} C_VEL
LIN {X 0,Y 418.239,Z 487.502,A -85,B 0,C 180,E1 -10127.768,E2 -10127.768} C_VEL
LIN {X 0,Y 418.256,Z 487.5,A -85,B 0,C 180,E1 -10130.619,E2 -10130.619} C_VEL
LIN {X 0,Y 418.241,Z 487.462,A -85,B 0,C 180,E1 -10133.977,E2 -10133.977} C_VEL
LIN {X 0,Y 418.257,Z 487.505,A -85,B 0,C 180,E1 -10137.157,E2 -10137.157} C_VEL
LIN {X 0,Y 418.285,Z 487.663,A -85,B 0,C 180,E1 -10138.54,E2 -10138.54} C_VEL
LIN {X 0,Y 420.783,Z 499.363,A -85,B 0,C 180,E1 -10141.575,E2 -10141.575} C_VEL
LIN {X 0,Y 421.833,Z 505.251,A -85,B 0,C 180,E1 -10143,E2 -10143} C_VEL
LIN {X 0,Y 421.234,Z 515.761,A -85,B 0,C 180,E1 -10145.348,E2 -10145.348} C_VEL
LIN {X 0,Y 420.723,Z 522.456,A -85,B 0,C 180,E1 -10146.84,E2 -10146.84} C_VEL
LIN {X 0,Y 425.012,Z 543.11,A -85,B 0,C 180,E1 -10147.487,E2 -10147.487} C_VEL
LIN {X 0,Y 426.97,Z 554.079,A -85,B 0,C 180,E1 -10147.79,E2 -10147.79} C_VEL
LIN {X 0,Y 425.397,Z 657.835,A -85,B 0,C 180,E1 -10149.574,E2 -10149.574} C_VEL
LIN {X 0,Y 425.014,Z 668.786,A -85,B 0,C 180,E1 -10149.87,E2 -10149.87} C_VEL
LIN {X 0,Y 424.493,Z 678.416,A -85,B 0,C 180,E1 -10150.223,E2 -10150.223} C_VEL
LIN {X 0,Y 423.914,Z 689.055,A -85,B 0,C 180,E1 -10150.731,E2 -10150.731} C_VEL
LIN {X 0,Y 423.197,Z 699.791,A -85,B 0,C 180,E1 -10151.374,E2 -10151.374} C_VEL
LIN {X 0,Y 422.49,Z 709.471,A -85,B 0,C 180,E1 -10152.077,E2 -10152.077} C_VEL
LIN {X 0,Y 421.657,Z 719.197,A -85,B 0,C 180,E1 -10152.917,E2 -10152.917} C_VEL
LIN {X 0,Y 420.776,Z 728.618,A -85,B 0,C 180,E1 -10153.879,E2 -10153.879} C_VEL
LIN {X 0,Y 419.983,Z 737.643,A -85,B 0,C 180,E1 -10154.967,E2 -10154.967} C_VEL
LIN {X 0,Y 419.376,Z 744.62,A -85,B 0,C 180,E1 -10155.937,E2 -10155.937} C_VEL
LIN {X 0,Y 418.781,Z 752.409,A -85,B 0,C 180,E1 -10157.201,E2 -10157.201} C_VEL
LIN {X 0,Y 418.195,Z 759.762,A -85,B 0,C 180,E1 -10158.611,E2 -10158.611} C_VEL
LIN {X 0,Y 417.776,Z 765.165,A -85,B 0,C 180,E1 -10159.826,E2 -10159.826} C_VEL
LIN {X 0,Y 417.447,Z 770.597,A -85,B 0,C 180,E1 -10161.285,E2 -10161.285} C_VEL
LIN {X 0,Y 417.25,Z 775.041,A -85,B 0,C 180,E1 -10162.743,E2 -10162.743} C_VEL
LIN {X 0,Y 417.113,Z 778.583,A -85,B 0,C 180,E1 -10164.198,E2 -10164.198} C_VEL
LIN {X 0,Y 417.079,Z 780.521,A -85,B 0,C 180,E1 -10165.167,E2 -10165.167} C_VEL
LIN {X 0,Y 417.023,Z 783.201,A -85,B 0,C 180,E1 -10167.102,E2 -10167.102} C_VEL
LIN {X 0,Y 417.009,Z 784.488,A -85,B 0,C 180,E1 -10169.034,E2 -10169.034} C_VEL
LIN {X 0,Y 417.003,Z 784.739,A -85,B 0,C 180,E1 -10170,E2 -10170} C_VEL
LIN {X 0,Y 417.054,Z 784.017,A -85,B 0,C 180,E1 -10171.931,E2 -10171.931} C_VEL
LIN {X 0,Y 417.023,Z 783.201,A -85,B 0,C 180,E1 -10172.898,E2 -10172.898} C_VEL
LIN {X 0,Y 417.077,Z 780.521,A -85,B 0,C 180,E1 -10174.833,E2 -10174.833} C_VEL
LIN {X 0,Y 417.227,Z 776.308,A -85,B 0,C 180,E1 -10176.771,E2 -10176.771} C_VEL
LIN {X 0,Y 417.343,Z 772.175,A -85,B 0,C 180,E1 -10178.229,E2 -10178.229} C_VEL
LIN {X 0,Y 417.669,Z 767.078,A -85,B 0,C 180,E1 -10179.687,E2 -10179.687} C_VEL
LIN {X 0,Y 418.101,Z 760.9,A -85,B 0,C 180,E1 -10181.146,E2 -10181.146} C_VEL
LIN {X 0,Y 418.561,Z 754.824,A -85,B 0,C 180,E1 -10182.361,E2 -10182.361} C_VEL
LIN {X 0,Y 419.087,Z 747.745,A -85,B 0,C 180,E1 -10183.578,E2 -10183.578} C_VEL
LIN {X 0,Y 419.819,Z 739.462,A -85,B 0,C 180,E1 -10184.791,E2 -10184.791} C_VEL
LIN {X 0,Y 420.601,Z 730.738,A -85,B 0,C 180,E1 -10185.879,E2 -10185.879} C_VEL
LIN {X 0,Y 421.388,Z 721.677,A -85,B 0,C 180,E1 -10186.845,E2 -10186.845} C_VEL
LIN {X 0,Y 422.238,Z 712.4,A -85,B 0,C 180,E1 -10187.683,E2 -10187.683} C_VEL
LIN {X 0,Y 422.98,Z 703.056,A -85,B 0,C 180,E1 -10188.402,E2 -10188.402} C_VEL
LIN {X 0,Y 423.654,Z 692.728,A -85,B 0,C 180,E1 -10189.066,E2 -10189.066} C_VEL
LIN {X 0,Y 424.339,Z 681.137,A -85,B 0,C 180,E1 -10189.658,E2 -10189.658} C_VEL
LIN {X 0,Y 424.942,Z 669.698,A -85,B 0,C 180,E1 -10190.102,E2 -10190.102} C_VEL
LIN {X 0,Y 425.376,Z 659.195,A -85,B 0,C 180,E1 -10190.396,E2 -10190.396} C_VEL
LIN {X 0,Y 425.929,Z 629.083,A -85,B 0,C 180,E1 -10190.936,E2 -10190.936} C_VEL
LIN {X 0,Y 426.897,Z 552.839,A -85,B 0,C 180,E1 -10192.236,E2 -10192.236} C_VEL
LIN {X 0,Y 420.759,Z 522.718,A -85,B 0,C 180,E1 -10193.138,E2 -10193.138} C_VEL
LIN {X 0,Y 420.735,Z 521.804,A -85,B 0,C 180,E1 -10193.259,E2 -10193.259} C_VEL
LIN {X 0,Y 421.859,Z 507.752,A -85,B 0,C 180,E1 -10196.464,E2 -10196.464} C_VEL
LIN {X 0,Y 421.531,Z 503.147,A -85,B 0,C 180,E1 -10197.558,E2 -10197.558} C_VEL
LIN {X 0,Y 418.977,Z 490.742,A -85,B 0,C 180,E1 -10200.636,E2 -10200.636} C_VEL
LIN {X 0,Y 418.258,Z 487.549,A -85,B 0,C 180,E1 -10201.532,E2 -10201.532} C_VEL
LIN {X 0,Y 418.258,Z 487.481,A -85,B 0,C 180,E1 -10204.84,E2 -10204.84} C_VEL
LIN {X 0,Y 418.255,Z 487.485,A -85,B 0,C 180,E1 -10208.44,E2 -10208.44} C_VEL
LIN {X 0,Y 418.222,Z 487.517,A -85,B 0,C 180,E1 -10210.947,E2 -10210.947} C_VEL
LIN {X 0,Y 418.213,Z 487.499,A -85,B 0,C 180,E1 -10213.729,E2 -10213.729} C_VEL
LIN {X 0,Y 418.205,Z 487.515,A -85,B 0,C 180,E1 -10216.448,E2 -10216.448} C_VEL
LIN {X 0,Y 418.262,Z 487.507,A -85,B 0,C 180,E1 -10219.123,E2 -10219.123} C_VEL
LIN {X 0,Y 418.233,Z 487.503,A -85,B 0,C 180,E1 -10222.164,E2 -10222.164} C_VEL
LIN {X 0,Y 418.261,Z 487.506,A -85,B 0,C 180,E1 -10225.419,E2 -10225.419} C_VEL
LIN {X 0,Y 418.206,Z 487.511,A -85,B 0,C 180,E1 -10228.603,E2 -10228.603} C_VEL
LIN {X 0,Y 418.286,Z 487.494,A -85,B 0,C 180,E1 -10231.936,E2 -10231.936} C_VEL
LIN {X 0,Y 418.284,Z 487.505,A -85,B 0,C 180,E1 -10235.162,E2 -10235.162} C_VEL
LIN {X 0,Y 418.227,Z 487.502,A -85,B 0,C 180,E1 -10238.303,E2 -10238.303} C_VEL
LIN {X 0,Y 418.276,Z 487.503,A -85,B 0,C 180,E1 -10241.382,E2 -10241.382} C_VEL
LIN {X 0,Y 418.294,Z 487.498,A -85,B 0,C 180,E1 -10244.405,E2 -10244.405} C_VEL
LIN {X 0,Y 418.347,Z 487.483,A -85,B 0,C 180,E1 -10247.385,E2 -10247.385} C_VEL
LIN {X 0,Y 418.333,Z 487.498,A -85,B 0,C 180,E1 -10250.328,E2 -10250.328} C_VEL
LIN {X 0,Y 418.485,Z 487.468,A -85,B 0,C 180,E1 -10253.248,E2 -10253.248} C_VEL
LIN {X 0,Y 418.333,Z 487.482,A -85,B 0,C 180,E1 -10255.181,E2 -10255.181} C_VEL
LIN {X 0,Y 418.536,Z 487.472,A -85,B 0,C 180,E1 -10258.075,E2 -10258.075} C_VEL
LIN {X 0,Y 418.663,Z 487.449,A -85,B 0,C 180,E1 -10260,E2 -10260} C_VEL
LIN {X 0,Y 418.503,Z 487.459,A -85,B 0,C 180,E1 -10262.887,E2 -10262.887} C_VEL
LIN {X 0,Y 418.483,Z 487.477,A -85,B 0,C 180,E1 -10266.751,E2 -10266.751} C_VEL
LIN {X 0,Y 418.333,Z 487.483,A -85,B 0,C 180,E1 -10269.671,E2 -10269.671} C_VEL
LIN {X 0,Y 418.337,Z 487.497,A -85,B 0,C 180,E1 -10273,E2 -10273} C_VEL
LIN {X 0,Y 418.303,Z 487.49,A -85,B 0,C 180,E1 -10276.735,E2 -10276.735} C_VEL
LIN {X 0,Y 418.262,Z 487.509,A -85,B 0,C 180,E1 -10279.79,E2 -10279.79} C_VEL
LIN {X 0,Y 418.229,Z 487.506,A -85,B 0,C 180,E1 -10282.736,E2 -10282.736} C_VEL
LIN {X 0,Y 418.262,Z 487.506,A -85,B 0,C 180,E1 -10285.904,E2 -10285.904} C_VEL
LIN {X 0,Y 418.266,Z 487.506,A -85,B 0,C 180,E1 -10289.161,E2 -10289.161} C_VEL
LIN {X 0,Y 418.251,Z 487.507,A -85,B 0,C 180,E1 -10292.845,E2 -10292.845} C_VEL
LIN {X 0,Y 418.24,Z 487.504,A -85,B 0,C 180,E1 -10296.239,E2 -10296.239} C_VEL
LIN {X 0,Y 418.247,Z 487.509,A -85,B 0,C 180,E1 -10299.682,E2 -10299.682} C_VEL
LIN {X 0,Y 418.276,Z 487.507,A -85,B 0,C 180,E1 -10302.33,E2 -10302.33} C_VEL
LIN {X 0,Y 418.267,Z 487.498,A -85,B 0,C 180,E1 -10305.114,E2 -10305.114} C_VEL
LIN {X 0,Y 418.285,Z 487.479,A -85,B 0,C 180,E1 -10307.774,E2 -10307.774} C_VEL
LIN {X 0,Y 418.261,Z 487.504,A -85,B 0,C 180,E1 -10311.56,E2 -10311.56} C_VEL
LIN {X 0,Y 418.253,Z 487.507,A -85,B 0,C 180,E1 -10315.159,E2 -10315.159} C_VEL
LIN {X 0,Y 418.24,Z 487.514,A -85,B 0,C 180,E1 -10317.472,E2 -10317.472} C_VEL
LIN {X 0,Y 418.271,Z 487.508,A -85,B 0,C 180,E1 -10320.894,E2 -10320.894} C_VEL
LIN {X 0,Y 418.266,Z 487.511,A -85,B 0,C 180,E1 -10324.096,E2 -10324.096} C_VEL
LIN {X 0,Y 418.233,Z 487.514,A -85,B 0,C 180,E1 -10327.264,E2 -10327.264} C_VEL
LIN {X 0,Y 418.279,Z 487.509,A -85,B 0,C 180,E1 -10330.364,E2 -10330.364} C_VEL
LIN {X 0,Y 418.313,Z 487.505,A -85,B 0,C 180,E1 -10333.405,E2 -10333.405} C_VEL
LIN {X 0,Y 418.342,Z 487.501,A -85,B 0,C 180,E1 -10336.999,E2 -10336.999} C_VEL
LIN {X 0,Y 418.337,Z 487.503,A -85,B 0,C 180,E1 -10340.329,E2 -10340.329} C_VEL
LIN {X 0,Y 418.509,Z 487.481,A -85,B 0,C 180,E1 -10342.28,E2 -10342.28} C_VEL
LIN {X 0,Y 418.509,Z 487.482,A -85,B 0,C 180,E1 -10344.217,E2 -10344.217} C_VEL
LIN {X 0,Y 418.541,Z 487.478,A -85,B 0,C 180,E1 -10348.076,E2 -10348.076} C_VEL
LIN {X 0,Y 418.669,Z 487.462,A -85,B 0,C 180,E1 -10350,E2 -10350} C_VEL
LIN {X 0,Y 418.507,Z 487.481,A -85,B 0,C 180,E1 -10352.888,E2 -10352.888} C_VEL
LIN {X 0,Y 418.49,Z 487.483,A -85,B 0,C 180,E1 -10356.751,E2 -10356.751} C_VEL
LIN {X 0,Y 418.353,Z 487.498,A -85,B 0,C 180,E1 -10359.155,E2 -10359.155} C_VEL
LIN {X 0,Y 418.351,Z 487.5,A -85,B 0,C 180,E1 -10362.614,E2 -10362.614} C_VEL
LIN {X 0,Y 418.318,Z 487.503,A -85,B 0,C 180,E1 -10363.345,E2 -10363.345} C_VEL
LIN {X 0,Y 417.625,Z 487.592,A -85,B 0,C 180,E1 -10364.148,E2 -10364.148} C_VEL
LIN {X 0,Y 414.746,Z 487.949,A -85,B 0,C 180,E1 -10365.454,E2 -10365.454} C_VEL
LIN {X 0,Y 412.333,Z 488.25,A -85,B 0,C 180,E1 -10366.508,E2 -10366.508} C_VEL
LIN {X 0,Y 411.312,Z 488.377,A -85,B 0,C 180,E1 -10367.323,E2 -10367.323} C_VEL
LIN {X 0,Y 411.236,Z 488.385,A -85,B 0,C 180,E1 -10367.599,E2 -10367.599} C_VEL
LIN {X 0,Y 411.192,Z 488.39,A -85,B 0,C 180,E1 -10371.034,E2 -10371.034} C_VEL
LIN {X 0,Y 411.222,Z 488.389,A -85,B 0,C 180,E1 -10374.215,E2 -10374.215} C_VEL
LIN {X 0,Y 411.254,Z 488.383,A -85,B 0,C 180,E1 -10377.477,E2 -10377.477} C_VEL
LIN {X 0,Y 411.192,Z 488.39,A -85,B 0,C 180,E1 -10380.847,E2 -10380.847} C_VEL
LIN {X 0,Y 411.2,Z 488.39,A -85,B 0,C 180,E1 -10384.333,E2 -10384.333} C_VEL
LIN {X 0,Y 411.198,Z 488.376,A -85,B 0,C 180,E1 -10387.972,E2 -10387.972} C_VEL
LIN {X 0,Y 411.203,Z 488.381,A -85,B 0,C 180,E1 -10391.236,E2 -10391.236} C_VEL
LIN {X 0,Y 411.225,Z 488.364,A -85,B 0,C 180,E1 -10394.482,E2 -10394.482} C_VEL
LIN {X 0,Y 411.224,Z 488.384,A -85,B 0,C 180,E1 -10397.296,E2 -10397.296} C_VEL
LIN {X 0,Y 411.216,Z 488.387,A -85,B 0,C 180,E1 -10400.776,E2 -10400.776} C_VEL
LIN {X 0,Y 411.191,Z 488.383,A -85,B 0,C 180,E1 -10404.471,E2 -10404.471} C_VEL
LIN {X 0,Y 411.163,Z 488.392,A -85,B 0,C 180,E1 -10408.003,E2 -10408.003} C_VEL
LIN {X 0,Y 411.215,Z 488.382,A -85,B 0,C 180,E1 -10411.41,E2 -10411.41} C_VEL
LIN {X 0,Y 411.228,Z 488.372,A -85,B 0,C 180,E1 -10414.707,E2 -10414.707} C_VEL
LIN {X 0,Y 411.196,Z 488.384,A -85,B 0,C 180,E1 -10417.914,E2 -10417.914} C_VEL
LIN {X 0,Y 411.215,Z 488.377,A -85,B 0,C 180,E1 -10421.052,E2 -10421.052} C_VEL
LIN {X 0,Y 411.245,Z 488.373,A -85,B 0,C 180,E1 -10424.132,E2 -10424.132} C_VEL
LIN {X 0,Y 411.294,Z 488.373,A -85,B 0,C 180,E1 -10427.166,E2 -10427.166} C_VEL
LIN {X 0,Y 411.285,Z 488.36,A -85,B 0,C 180,E1 -10430.162,E2 -10430.162} C_VEL
LIN {X 0,Y 411.449,Z 488.354,A -85,B 0,C 180,E1 -10433.133,E2 -10433.133} C_VEL
LIN {X 0,Y 411.309,Z 488.369,A -85,B 0,C 180,E1 -10435.099,E2 -10435.099} C_VEL
LIN {X 0,Y 411.505,Z 488.329,A -85,B 0,C 180,E1 -10438.043,E2 -10438.043} C_VEL
LIN {X 0,Y 411.633,Z 488.325,A -85,B 0,C 180,E1 -10440,E2 -10440} C_VEL
LIN {X 0,Y 411.458,Z 488.351,A -85,B 0,C 180,E1 -10442.938,E2 -10442.938} C_VEL
LIN {X 0,Y 411.452,Z 488.345,A -85,B 0,C 180,E1 -10446.868,E2 -10446.868} C_VEL
LIN {X 0,Y 411.285,Z 488.376,A -85,B 0,C 180,E1 -10449.839,E2 -10449.839} C_VEL
LIN {X 0,Y 411.297,Z 488.356,A -85,B 0,C 180,E1 -10453.105,E2 -10453.105} C_VEL
LIN {X 0,Y 411.25,Z 488.383,A -85,B 0,C 180,E1 -10456.889,E2 -10456.889} C_VEL
LIN {X 0,Y 411.224,Z 488.374,A -85,B 0,C 180,E1 -10459.988,E2 -10459.988} C_VEL
LIN {X 0,Y 411.19,Z 488.389,A -85,B 0,C 180,E1 -10463.149,E2 -10463.149} C_VEL
LIN {X 0,Y 411.232,Z 488.376,A -85,B 0,C 180,E1 -10466.382,E2 -10466.382} C_VEL
LIN {X 0,Y 411.195,Z 488.387,A -85,B 0,C 180,E1 -10469.714,E2 -10469.714} C_VEL
LIN {X 0,Y 411.201,Z 488.378,A -85,B 0,C 180,E1 -10473.157,E2 -10473.157} C_VEL
LIN {X 0,Y 411.191,Z 488.391,A -85,B 0,C 180,E1 -10476.554,E2 -10476.554} C_VEL
LIN {X 0,Y 411.223,Z 488.385,A -85,B 0,C 180,E1 -10479.731,E2 -10479.731} C_VEL
LIN {X 0,Y 411.173,Z 488.395,A -85,B 0,C 180,E1 -10483.134,E2 -10483.134} C_VEL
LIN {X 0,Y 411.169,Z 488.381,A -85,B 0,C 180,E1 -10485.881,E2 -10485.881} C_VEL
LIN {X 0,Y 411.163,Z 488.393,A -85,B 0,C 180,E1 -10488.772,E2 -10488.772} C_VEL
LIN {X 0,Y 411.205,Z 488.354,A -85,B 0,C 180,E1 -10491.832,E2 -10491.832} C_VEL
LIN {X 0,Y 411.209,Z 488.356,A -85,B 0,C 180,E1 -10495.122,E2 -10495.122} C_VEL
LIN {X 0,Y 411.228,Z 488.526,A -85,B 0,C 180,E1 -10498.197,E2 -10498.197} C_VEL
LIN {X 0,Y 413.495,Z 499.151,A -85,B 0,C 180,E1 -10501.027,E2 -10501.027} C_VEL
LIN {X 0,Y 414.934,Z 507.395,A -85,B 0,C 180,E1 -10503.059,E2 -10503.059} C_VEL
LIN {X 0,Y 414.091,Z 518.897,A -85,B 0,C 180,E1 -10505.697,E2 -10505.697} C_VEL
LIN {X 0,Y 413.877,Z 522.295,A -85,B 0,C 180,E1 -10506.438,E2 -10506.438} C_VEL
LIN {X 0,Y 419.648,Z 550.403,A -85,B 0,C 180,E1 -10507.318,E2 -10507.318} C_VEL
LIN {X 0,Y 420.392,Z 555.004,A -85,B 0,C 180,E1 -10507.444,E2 -10507.444} C_VEL
LIN {X 0,Y 418.763,Z 657.637,A -85,B 0,C 180,E1 -10509.236,E2 -10509.236} C_VEL
LIN {X 0,Y 418.363,Z 668.589,A -85,B 0,C 180,E1 -10509.536,E2 -10509.536} C_VEL
LIN {X 0,Y 417.735,Z 679.579,A -85,B 0,C 180,E1 -10509.954,E2 -10509.954} C_VEL
LIN {X 0,Y 417.194,Z 689.045,A -85,B 0,C 180,E1 -10510.42,E2 -10510.42} C_VEL
LIN {X 0,Y 416.448,Z 699.623,A -85,B 0,C 180,E1 -10511.063,E2 -10511.063} C_VEL
LIN {X 0,Y 415.716,Z 709.272,A -85,B 0,C 180,E1 -10511.775,E2 -10511.775} C_VEL
LIN {X 0,Y 414.848,Z 718.998,A -85,B 0,C 180,E1 -10512.628,E2 -10512.628} C_VEL
LIN {X 0,Y 413.934,Z 728.419,A -85,B 0,C 180,E1 -10513.605,E2 -10513.605} C_VEL
LIN {X 0,Y 413.076,Z 737.443,A -85,B 0,C 180,E1 -10514.71,E2 -10514.71} C_VEL
LIN {X 0,Y 412.431,Z 744.421,A -85,B 0,C 180,E1 -10515.695,E2 -10515.695} C_VEL
LIN {X 0,Y 411.84,Z 751.971,A -85,B 0,C 180,E1 -10516.936,E2 -10516.936} C_VEL
LIN {X 0,Y 411.318,Z 758.426,A -85,B 0,C 180,E1 -10518.169,E2 -10518.169} C_VEL
LIN {X 0,Y 410.72,Z 764.965,A -85,B 0,C 180,E1 -10519.65,E2 -10519.65} C_VEL
LIN {X 0,Y 410.374,Z 770.397,A -85,B 0,C 180,E1 -10521.134,E2 -10521.134} C_VEL
LIN {X 0,Y 410.162,Z 774.842,A -85,B 0,C 180,E1 -10522.617,E2 -10522.617} C_VEL
LIN {X 0,Y 410.036,Z 778.384,A -85,B 0,C 180,E1 -10524.097,E2 -10524.097} C_VEL
LIN {X 0,Y 409.989,Z 780.323,A -85,B 0,C 180,E1 -10525.083,E2 -10525.083} C_VEL
LIN {X 0,Y 409.921,Z 783.002,A -85,B 0,C 180,E1 -10527.052,E2 -10527.052} C_VEL
LIN {X 0,Y 409.934,Z 784.29,A -85,B 0,C 180,E1 -10529.018,E2 -10529.018} C_VEL
LIN {X 0,Y 409.925,Z 784.542,A -85,B 0,C 180,E1 -10530,E2 -10530} C_VEL
LIN {X 0,Y 409.964,Z 783.819,A -85,B 0,C 180,E1 -10531.965,E2 -10531.965} C_VEL
LIN {X 0,Y 409.921,Z 783.002,A -85,B 0,C 180,E1 -10532.948,E2 -10532.948} C_VEL
LIN {X 0,Y 409.988,Z 780.323,A -85,B 0,C 180,E1 -10534.917,E2 -10534.917} C_VEL
LIN {X 0,Y 410.058,Z 777.71,A -85,B 0,C 180,E1 -10536.244,E2 -10536.244} C_VEL
LIN {X 0,Y 410.193,Z 773.543,A -85,B 0,C 180,E1 -10537.878,E2 -10537.878} C_VEL
LIN {X 0,Y 410.504,Z 768.783,A -85,B 0,C 180,E1 -10539.36,E2 -10539.36} C_VEL
LIN {X 0,Y 410.98,Z 761.838,A -85,B 0,C 180,E1 -10541.092,E2 -10541.092} C_VEL
LIN {X 0,Y 411.503,Z 755.963,A -85,B 0,C 180,E1 -10542.326,E2 -10542.326} C_VEL
LIN {X 0,Y 412.153,Z 747.546,A -85,B 0,C 180,E1 -10543.811,E2 -10543.811} C_VEL
LIN {X 0,Y 412.902,Z 739.262,A -85,B 0,C 180,E1 -10545.044,E2 -10545.044} C_VEL
LIN {X 0,Y 413.707,Z 730.538,A -85,B 0,C 180,E1 -10546.151,E2 -10546.151} C_VEL
LIN {X 0,Y 414.565,Z 721.478,A -85,B 0,C 180,E1 -10547.13,E2 -10547.13} C_VEL
LIN {X 0,Y 415.462,Z 712.202,A -85,B 0,C 180,E1 -10547.982,E2 -10547.982} C_VEL
LIN {X 0,Y 416.233,Z 702.858,A -85,B 0,C 180,E1 -10548.712,E2 -10548.712} C_VEL
LIN {X 0,Y 416.966,Z 692.03,A -85,B 0,C 180,E1 -10549.413,E2 -10549.413} C_VEL
LIN {X 0,Y 417.637,Z 680.938,A -85,B 0,C 180,E1 -10549.987,E2 -10549.987} C_VEL
LIN {X 0,Y 418.245,Z 670.412,A -85,B 0,C 180,E1 -10550.406,E2 -10550.406} C_VEL
LIN {X 0,Y 418.724,Z 658.997,A -85,B 0,C 180,E1 -10550.734,E2 -10550.734} C_VEL
LIN {X 0,Y 419.304,Z 628.885,A -85,B 0,C 180,E1 -10551.283,E2 -10551.283} C_VEL
LIN {X 0,Y 420.23,Z 553.445,A -85,B 0,C 180,E1 -10552.594,E2 -10552.594} C_VEL
LIN {X 0,Y 413.93,Z 522.746,A -85,B 0,C 180,E1 -10553.53,E2 -10553.53} C_VEL
LIN {X 0,Y 413.872,Z 521.45,A -85,B 0,C 180,E1 -10553.698,E2 -10553.698} C_VEL
LIN {X 0,Y 415.006,Z 507.547,A -85,B 0,C 180,E1 -10556.936,E2 -10556.936} C_VEL
LIN {X 0,Y 413.597,Z 499.454,A -85,B 0,C 180,E1 -10558.965,E2 -10558.965} C_VEL
LIN {X 0,Y 411.232,Z 488.549,A -85,B 0,C 180,E1 -10561.803,E2 -10561.803} C_VEL
LIN {X 0,Y 411.209,Z 488.356,A -85,B 0,C 180,E1 -10564.878,E2 -10564.878} C_VEL
LIN {X 0,Y 411.205,Z 488.354,A -85,B 0,C 180,E1 -10568.168,E2 -10568.168} C_VEL
LIN {X 0,Y 411.163,Z 488.393,A -85,B 0,C 180,E1 -10571.228,E2 -10571.228} C_VEL
LIN {X 0,Y 411.176,Z 488.38,A -85,B 0,C 180,E1 -10574.489,E2 -10574.489} C_VEL
LIN {X 0,Y 411.195,Z 488.382,A -85,B 0,C 180,E1 -10578.196,E2 -10578.196} C_VEL
LIN {X 0,Y 411.226,Z 488.385,A -85,B 0,C 180,E1 -10580.776,E2 -10580.776} C_VEL
LIN {X 0,Y 411.195,Z 488.387,A -85,B 0,C 180,E1 -10584.471,E2 -10584.471} C_VEL
LIN {X 0,Y 411.202,Z 488.378,A -85,B 0,C 180,E1 -10586.872,E2 -10586.872} C_VEL
LIN {X 0,Y 411.227,Z 488.383,A -85,B 0,C 180,E1 -10590.643,E2 -10590.643} C_VEL
LIN {X 0,Y 411.232,Z 488.376,A -85,B 0,C 180,E1 -10593.618,E2 -10593.618} C_VEL
LIN {X 0,Y 411.19,Z 488.389,A -85,B 0,C 180,E1 -10596.851,E2 -10596.851} C_VEL
LIN {X 0,Y 411.208,Z 488.377,A -85,B 0,C 180,E1 -10600.05,E2 -10600.05} C_VEL
LIN {X 0,Y 411.256,Z 488.383,A -85,B 0,C 180,E1 -10603.13,E2 -10603.13} C_VEL
LIN {X 0,Y 411.297,Z 488.356,A -85,B 0,C 180,E1 -10606.895,E2 -10606.895} C_VEL
LIN {X 0,Y 411.285,Z 488.376,A -85,B 0,C 180,E1 -10610.161,E2 -10610.161} C_VEL
LIN {X 0,Y 411.452,Z 488.345,A -85,B 0,C 180,E1 -10613.132,E2 -10613.132} C_VEL
LIN {X 0,Y 411.304,Z 488.356,A -85,B 0,C 180,E1 -10615.098,E2 -10615.098} C_VEL
LIN {X 0,Y 411.505,Z 488.348,A -85,B 0,C 180,E1 -10618.042,E2 -10618.042} C_VEL
LIN {X 0,Y 411.633,Z 488.325,A -85,B 0,C 180,E1 -10620,E2 -10620} C_VEL
LIN {X 0,Y 411.458,Z 488.336,A -85,B 0,C 180,E1 -10622.937,E2 -10622.937} C_VEL
LIN {X 0,Y 411.447,Z 488.354,A -85,B 0,C 180,E1 -10626.867,E2 -10626.867} C_VEL
LIN {X 0,Y 411.285,Z 488.36,A -85,B 0,C 180,E1 -10629.838,E2 -10629.838} C_VEL
LIN {X 0,Y 411.296,Z 488.374,A -85,B 0,C 180,E1 -10633.104,E2 -10633.104} C_VEL
LIN {X 0,Y 411.248,Z 488.369,A -85,B 0,C 180,E1 -10636.889,E2 -10636.889} C_VEL
LIN {X 0,Y 411.221,Z 488.386,A -85,B 0,C 180,E1 -10639.987,E2 -10639.987} C_VEL
LIN {X 0,Y 411.194,Z 488.383,A -85,B 0,C 180,E1 -10643.147,E2 -10643.147} C_VEL
LIN {X 0,Y 411.229,Z 488.382,A -85,B 0,C 180,E1 -10646.381,E2 -10646.381} C_VEL
LIN {X 0,Y 411.202,Z 488.378,A -85,B 0,C 180,E1 -10649.712,E2 -10649.712} C_VEL
LIN {X 0,Y 411.198,Z 488.388,A -85,B 0,C 180,E1 -10653.156,E2 -10653.156} C_VEL
LIN {X 0,Y 411.187,Z 488.383,A -85,B 0,C 180,E1 -10656.553,E2 -10656.553} C_VEL
LIN {X 0,Y 411.211,Z 488.384,A -85,B 0,C 180,E1 -10659.729,E2 -10659.729} C_VEL
LIN {X 0,Y 411.223,Z 488.386,A -85,B 0,C 180,E1 -10663.126,E2 -10663.126} C_VEL
LIN {X 0,Y 411.223,Z 488.358,A -85,B 0,C 180,E1 -10665.872,E2 -10665.872} C_VEL
LIN {X 0,Y 411.204,Z 488.381,A -85,B 0,C 180,E1 -10668.764,E2 -10668.764} C_VEL
LIN {X 0,Y 411.199,Z 488.376,A -85,B 0,C 180,E1 -10672.028,E2 -10672.028} C_VEL
LIN {X 0,Y 411.2,Z 488.39,A -85,B 0,C 180,E1 -10675.667,E2 -10675.667} C_VEL
LIN {X 0,Y 411.192,Z 488.39,A -85,B 0,C 180,E1 -10679.153,E2 -10679.153} C_VEL
LIN {X 0,Y 411.254,Z 488.383,A -85,B 0,C 180,E1 -10682.523,E2 -10682.523} C_VEL
LIN {X 0,Y 411.222,Z 488.389,A -85,B 0,C 180,E1 -10685.785,E2 -10685.785} C_VEL
LIN {X 0,Y 411.192,Z 488.39,A -85,B 0,C 180,E1 -10688.966,E2 -10688.966} C_VEL
LIN {X 0,Y 411.248,Z 488.386,A -85,B 0,C 180,E1 -10692.085,E2 -10692.085} C_VEL
LIN {X 0,Y 411.256,Z 488.384,A -85,B 0,C 180,E1 -10695.148,E2 -10695.148} C_VEL
LIN {X 0,Y 411.28,Z 488.381,A -85,B 0,C 180,E1 -10698.167,E2 -10698.167} C_VEL
LIN {X 0,Y 411.478,Z 488.356,A -85,B 0,C 180,E1 -10702.147,E2 -10702.147} C_VEL
LIN {X 0,Y 411.471,Z 488.358,A -85,B 0,C 180,E1 -10704.118,E2 -10704.118} C_VEL
LIN {X 0,Y 411.51,Z 488.354,A -85,B 0,C 180,E1 -10708.043,E2 -10708.043} C_VEL
LIN {X 0,Y 411.639,Z 488.338,A -85,B 0,C 180,E1 -10710,E2 -10710} C_VEL
LIN {X 0,Y 411.462,Z 488.359,A -85,B 0,C 180,E1 -10712.937,E2 -10712.937} C_VEL
LIN {X 0,Y 411.457,Z 488.359,A -85,B 0,C 180,E1 -10716.867,E2 -10716.867} C_VEL
LIN {X 0,Y 411.289,Z 488.38,A -85,B 0,C 180,E1 -10719.839,E2 -10719.839} C_VEL
LIN {X 0,Y 411.278,Z 488.38,A -85,B 0,C 180,E1 -10723.333,E2 -10723.333} C_VEL
LIN {X 0,Y 411.253,Z 488.384,A -85,B 0,C 180,E1 -10726.889,E2 -10726.889} C_VEL
LIN {X 0,Y 411.236,Z 488.385,A -85,B 0,C 180,E1 -10727.599,E2 -10727.599} C_VEL
LIN {X 0,Y 410.576,Z 488.47,A -85,B 0,C 180,E1 -10728.416,E2 -10728.416} C_VEL
LIN {X 0,Y 407.688,Z 488.829,A -85,B 0,C 180,E1 -10729.745,E2 -10729.745} C_VEL
LIN {X 0,Y 405.243,Z 489.132,A -85,B 0,C 180,E1 -10730.817,E2 -10730.817} C_VEL
LIN {X 0,Y 404.207,Z 489.262,A -85,B 0,C 180,E1 -10731.647,E2 -10731.647} C_VEL
LIN {X 0,Y 404.131,Z 489.269,A -85,B 0,C 180,E1 -10731.928,E2 -10731.928} C_VEL
LIN {X 0,Y 404.211,Z 489.261,A -85,B 0,C 180,E1 -10735.296,E2 -10735.296} C_VEL
LIN {X 0,Y 404.192,Z 489.265,A -85,B 0,C 180,E1 -10737.999,E2 -10737.999} C_VEL
LIN {X 0,Y 404.137,Z 489.27,A -85,B 0,C 180,E1 -10741.559,E2 -10741.559} C_VEL
LIN {X 0,Y 404.179,Z 489.259,A -85,B 0,C 180,E1 -10745.016,E2 -10745.016} C_VEL
LIN {X 0,Y 404.157,Z 489.266,A -85,B 0,C 180,E1 -10748.756,E2 -10748.756} C_VEL
LIN {X 0,Y 404.185,Z 489.246,A -85,B 0,C 180,E1 -10751.61,E2 -10751.61} C_VEL
LIN {X 0,Y 404.19,Z 489.241,A -85,B 0,C 180,E1 -10754.529,E2 -10754.529} C_VEL
LIN {X 0,Y 404.202,Z 489.259,A -85,B 0,C 180,E1 -10757.305,E2 -10757.305} C_VEL
LIN {X 0,Y 404.161,Z 489.258,A -85,B 0,C 180,E1 -10759.955,E2 -10759.955} C_VEL
LIN {X 0,Y 404.131,Z 489.261,A -85,B 0,C 180,E1 -10763.124,E2 -10763.124} C_VEL
LIN {X 0,Y 404.137,Z 489.269,A -85,B 0,C 180,E1 -10766.188,E2 -10766.188} C_VEL
LIN {X 0,Y 404.146,Z 489.252,A -85,B 0,C 180,E1 -10769.716,E2 -10769.716} C_VEL
LIN {X 0,Y 404.186,Z 489.259,A -85,B 0,C 180,E1 -10773.123,E2 -10773.123} C_VEL
LIN {X 0,Y 404.168,Z 489.248,A -85,B 0,C 180,E1 -10775.334,E2 -10775.334} C_VEL
LIN {X 0,Y 404.15,Z 489.269,A -85,B 0,C 180,E1 -10778.582,E2 -10778.582} C_VEL
LIN {X 0,Y 404.201,Z 489.249,A -85,B 0,C 180,E1 -10781.762,E2 -10781.762} C_VEL
LIN {X 0,Y 404.196,Z 489.26,A -85,B 0,C 180,E1 -10784.882,E2 -10784.882} C_VEL
LIN {X 0,Y 404.247,Z 489.252,A -85,B 0,C 180,E1 -10787.959,E2 -10787.959} C_VEL
LIN {X 0,Y 404.393,Z 489.227,A -85,B 0,C 180,E1 -10792.133,E2 -10792.133} C_VEL
LIN {X 0,Y 404.428,Z 489.23,A -85,B 0,C 180,E1 -10794.016,E2 -10794.016} C_VEL
LIN {X 0,Y 404.474,Z 489.204,A -85,B 0,C 180,E1 -10798.009,E2 -10798.009} C_VEL
LIN {X 0,Y 404.602,Z 489.2,A -85,B 0,C 180,E1 -10800,E2 -10800} C_VEL
LIN {X 0,Y 404.416,Z 489.228,A -85,B 0,C 180,E1 -10802.989,E2 -10802.989} C_VEL
LIN {X 0,Y 404.399,Z 489.225,A -85,B 0,C 180,E1 -10806.988,E2 -10806.988} C_VEL
LIN {X 0,Y 404.25,Z 489.254,A -85,B 0,C 180,E1 -10810.012,E2 -10810.012} C_VEL
LIN {X 0,Y 404.259,Z 489.231,A -85,B 0,C 180,E1 -10813.212,E2 -10813.212} C_VEL
LIN {X 0,Y 404.209,Z 489.259,A -85,B 0,C 180,E1 -10817.008,E2 -10817.008} C_VEL
LIN {X 0,Y 404.157,Z 489.251,A -85,B 0,C 180,E1 -10820.352,E2 -10820.352} C_VEL
LIN {X 0,Y 404.157,Z 489.263,A -85,B 0,C 180,E1 -10823.576,E2 -10823.576} C_VEL
LIN {X 0,Y 404.178,Z 489.257,A -85,B 0,C 180,E1 -10825.767,E2 -10825.767} C_VEL
LIN {X 0,Y 404.189,Z 489.249,A -85,B 0,C 180,E1 -10828,E2 -10828} C_VEL
LIN {X 0,Y 404.134,Z 489.263,A -85,B 0,C 180,E1 -10831.559,E2 -10831.559} C_VEL
LIN {X 0,Y 404.181,Z 489.265,A -85,B 0,C 180,E1 -10835.017,E2 -10835.017} C_VEL
LIN {X 0,Y 404.159,Z 489.262,A -85,B 0,C 180,E1 -10838.757,E2 -10838.757} C_VEL
LIN {X 0,Y 404.146,Z 489.261,A -85,B 0,C 180,E1 -10841.605,E2 -10841.605} C_VEL
LIN {X 0,Y 404.143,Z 489.269,A -85,B 0,C 180,E1 -10844.523,E2 -10844.523} C_VEL
LIN {X 0,Y 404.136,Z 489.252,A -85,B 0,C 180,E1 -10847.297,E2 -10847.297} C_VEL
LIN {X 0,Y 404.167,Z 489.264,A -85,B 0,C 180,E1 -10849.956,E2 -10849.956} C_VEL
LIN {X 0,Y 404.134,Z 489.213,A -85,B 0,C 180,E1 -10853.126,E2 -10853.126} C_VEL
LIN {X 0,Y 404.144,Z 489.268,A -85,B 0,C 180,E1 -10856.189,E2 -10856.189} C_VEL
LIN {X 0,Y 404.19,Z 489.447,A -85,B 0,C 180,E1 -10857.863,E2 -10857.863} C_VEL
LIN {X 0,Y 406.483,Z 500.12,A -85,B 0,C 180,E1 -10860.763,E2 -10860.763} C_VEL
LIN {X 0,Y 408.009,Z 508.368,A -85,B 0,C 180,E1 -10862.841,E2 -10862.841} C_VEL
LIN {X 0,Y 407.16,Z 519.787,A -85,B 0,C 180,E1 -10865.528,E2 -10865.528} C_VEL
LIN {X 0,Y 406.985,Z 521.97,A -85,B 0,C 180,E1 -10866.004,E2 -10866.004} C_VEL
LIN {X 0,Y 408.917,Z 530.84,A -85,B 0,C 180,E1 -10866.328,E2 -10866.328} C_VEL
LIN {X 0,Y 413.689,Z 554.684,A -85,B 0,C 180,E1 -10867.055,E2 -10867.055} C_VEL
LIN {X 0,Y 412.194,Z 656.08,A -85,B 0,C 180,E1 -10868.856,E2 -10868.856} C_VEL
LIN {X 0,Y 411.728,Z 667.478,A -85,B 0,C 180,E1 -10869.158,E2 -10869.158} C_VEL
LIN {X 0,Y 411.168,Z 678.021,A -85,B 0,C 180,E1 -10869.554,E2 -10869.554} C_VEL
LIN {X 0,Y 410.487,Z 689.04,A -85,B 0,C 180,E1 -10870.098,E2 -10870.098} C_VEL
LIN {X 0,Y 409.687,Z 699.424,A -85,B 0,C 180,E1 -10870.738,E2 -10870.738} C_VEL
LIN {X 0,Y 408.948,Z 709.073,A -85,B 0,C 180,E1 -10871.462,E2 -10871.462} C_VEL
LIN {X 0,Y 408.042,Z 718.799,A -85,B 0,C 180,E1 -10872.328,E2 -10872.328} C_VEL
LIN {X 0,Y 407.088,Z 728.22,A -85,B 0,C 180,E1 -10873.321,E2 -10873.321} C_VEL
LIN {X 0,Y 406.193,Z 737.244,A -85,B 0,C 180,E1 -10874.444,E2 -10874.444} C_VEL
LIN {X 0,Y 405.511,Z 744.221,A -85,B 0,C 180,E1 -10875.446,E2 -10875.446} C_VEL
LIN {X 0,Y 404.845,Z 752.078,A -85,B 0,C 180,E1 -10876.765,E2 -10876.765} C_VEL
LIN {X 0,Y 404.196,Z 759.364,A -85,B 0,C 180,E1 -10878.211,E2 -10878.211} C_VEL
LIN {X 0,Y 403.683,Z 764.765,A -85,B 0,C 180,E1 -10879.467,E2 -10879.467} C_VEL
LIN {X 0,Y 403.323,Z 770.198,A -85,B 0,C 180,E1 -10880.977,E2 -10880.977} C_VEL
LIN {X 0,Y 403.068,Z 774.642,A -85,B 0,C 180,E1 -10882.486,E2 -10882.486} C_VEL
LIN {X 0,Y 402.939,Z 778.185,A -85,B 0,C 180,E1 -10883.993,E2 -10883.993} C_VEL
LIN {X 0,Y 402.904,Z 780.124,A -85,B 0,C 180,E1 -10884.997,E2 -10884.997} C_VEL
LIN {X 0,Y 402.82,Z 782.804,A -85,B 0,C 180,E1 -10887,E2 -10887} C_VEL
LIN {X 0,Y 402.861,Z 784.093,A -85,B 0,C 180,E1 -10889,E2 -10889} C_VEL
LIN {X 0,Y 402.85,Z 784.344,A -85,B 0,C 180,E1 -10890,E2 -10890} C_VEL
LIN {X 0,Y 402.862,Z 783.621,A -85,B 0,C 180,E1 -10891.999,E2 -10891.999} C_VEL
LIN {X 0,Y 402.82,Z 782.804,A -85,B 0,C 180,E1 -10893,E2 -10893} C_VEL
LIN {X 0,Y 402.901,Z 780.124,A -85,B 0,C 180,E1 -10895.003,E2 -10895.003} C_VEL
LIN {X 0,Y 402.979,Z 777.75,A -85,B 0,C 180,E1 -10896.232,E2 -10896.232} C_VEL
LIN {X 0,Y 403.139,Z 773.345,A -85,B 0,C 180,E1 -10898.017,E2 -10898.017} C_VEL
LIN {X 0,Y 403.452,Z 768.583,A -85,B 0,C 180,E1 -10899.525,E2 -10899.525} C_VEL
LIN {X 0,Y 403.984,Z 761.639,A -85,B 0,C 180,E1 -10901.286,E2 -10901.286} C_VEL
LIN {X 0,Y 404.486,Z 755.763,A -85,B 0,C 180,E1 -10902.544,E2 -10902.544} C_VEL
LIN {X 0,Y 405.065,Z 748.699,A -85,B 0,C 180,E1 -10903.836,E2 -10903.836} C_VEL
LIN {X 0,Y 405.82,Z 740.882,A -85,B 0,C 180,E1 -10905.056,E2 -10905.056} C_VEL
LIN {X 0,Y 406.767,Z 731.4,A -85,B 0,C 180,E1 -10906.305,E2 -10906.305} C_VEL
LIN {X 0,Y 407.636,Z 722.52,A -85,B 0,C 180,E1 -10907.301,E2 -10907.301} C_VEL
LIN {X 0,Y 408.559,Z 713.468,A -85,B 0,C 180,E1 -10908.166,E2 -10908.166} C_VEL
LIN {X 0,Y 409.491,Z 702.659,A -85,B 0,C 180,E1 -10909.031,E2 -10909.031} C_VEL
LIN {X 0,Y 410.179,Z 692.985,A -85,B 0,C 180,E1 -10909.678,E2 -10909.678} C_VEL
LIN {X 0,Y 410.881,Z 682.1,A -85,B 0,C 180,E1 -10910.265,E2 -10910.265} C_VEL
LIN {X 0,Y 411.571,Z 670.213,A -85,B 0,C 180,E1 -10910.752,E2 -10910.752} C_VEL
LIN {X 0,Y 412.091,Z 658.799,A -85,B 0,C 180,E1 -10911.084,E2 -10911.084} C_VEL
LIN {X 0,Y 412.712,Z 628.688,A -85,B 0,C 180,E1 -10911.64,E2 -10911.64} C_VEL
LIN {X 0,Y 413.689,Z 554.751,A -85,B 0,C 180,E1 -10912.944,E2 -10912.944} C_VEL
LIN {X 0,Y 407.747,Z 525.54,A -85,B 0,C 180,E1 -10913.843,E2 -10913.843} C_VEL
LIN {X 0,Y 407.002,Z 521.954,A -85,B 0,C 180,E1 -10913.996,E2 -10913.996} C_VEL
LIN {X 0,Y 408.075,Z 509.638,A -85,B 0,C 180,E1 -10916.877,E2 -10916.877} C_VEL
LIN {X 0,Y 407.111,Z 502.984,A -85,B 0,C 180,E1 -10918.556,E2 -10918.556} C_VEL
LIN {X 0,Y 404.574,Z 491.145,A -85,B 0,C 180,E1 -10921.657,E2 -10921.657} C_VEL
LIN {X 0,Y 404.148,Z 489.281,A -85,B 0,C 180,E1 -10922.243,E2 -10922.243} C_VEL
LIN {X 0,Y 404.179,Z 489.222,A -85,B 0,C 180,E1 -10925.189,E2 -10925.189} C_VEL
LIN {X 0,Y 404.155,Z 489.246,A -85,B 0,C 180,E1 -10928.756,E2 -10928.756} C_VEL
LIN {X 0,Y 404.122,Z 489.265,A -85,B 0,C 180,E1 -10931.599,E2 -10931.599} C_VEL
LIN {X 0,Y 404.145,Z 489.256,A -85,B 0,C 180,E1 -10934.522,E2 -10934.522} C_VEL
LIN {X 0,Y 404.167,Z 489.262,A -85,B 0,C 180,E1 -10937.299,E2 -10937.299} C_VEL
LIN {X 0,Y 404.165,Z 489.264,A -85,B 0,C 180,E1 -10939.954,E2 -10939.954} C_VEL
LIN {X 0,Y 404.136,Z 489.264,A -85,B 0,C 180,E1 -10943.123,E2 -10943.123} C_VEL
LIN {X 0,Y 404.14,Z 489.258,A -85,B 0,C 180,E1 -10946.187,E2 -10946.187} C_VEL
LIN {X 0,Y 404.14,Z 489.268,A -85,B 0,C 180,E1 -10949.714,E2 -10949.714} C_VEL
LIN {X 0,Y 404.189,Z 489.248,A -85,B 0,C 180,E1 -10953.122,E2 -10953.122} C_VEL
LIN {X 0,Y 404.168,Z 489.265,A -85,B 0,C 180,E1 -10955.333,E2 -10955.333} C_VEL
LIN {X 0,Y 404.131,Z 489.257,A -85,B 0,C 180,E1 -10958.58,E2 -10958.58} C_VEL
LIN {X 0,Y 404.203,Z 489.26,A -85,B 0,C 180,E1 -10961.761,E2 -10961.761} C_VEL
LIN {X 0,Y 404.198,Z 489.256,A -85,B 0,C 180,E1 -10964.881,E2 -10964.881} C_VEL
LIN {X 0,Y 404.248,Z 489.248,A -85,B 0,C 180,E1 -10967.958,E2 -10967.958} C_VEL
LIN {X 0,Y 404.398,Z 489.228,A -85,B 0,C 180,E1 -10972.127,E2 -10972.127} C_VEL
LIN {X 0,Y 404.415,Z 489.211,A -85,B 0,C 180,E1 -10974.014,E2 -10974.014} C_VEL
LIN {X 0,Y 404.474,Z 489.224,A -85,B 0,C 180,E1 -10978.008,E2 -10978.008} C_VEL
LIN {X 0,Y 404.602,Z 489.2,A -85,B 0,C 180,E1 -10980,E2 -10980} C_VEL
LIN {X 0,Y 404.415,Z 489.213,A -85,B 0,C 180,E1 -10982.988,E2 -10982.988} C_VEL
LIN {X 0,Y 404.394,Z 489.234,A -85,B 0,C 180,E1 -10986.987,E2 -10986.987} C_VEL
LIN {X 0,Y 404.25,Z 489.235,A -85,B 0,C 180,E1 -10990.011,E2 -10990.011} C_VEL
LIN {X 0,Y 404.257,Z 489.252,A -85,B 0,C 180,E1 -10993.211,E2 -10993.211} C_VEL
LIN {X 0,Y 404.207,Z 489.244,A -85,B 0,C 180,E1 -10997.007,E2 -10997.007} C_VEL
LIN {X 0,Y 404.155,Z 489.264,A -85,B 0,C 180,E1 -11000.351,E2 -11000.351} C_VEL
LIN {X 0,Y 404.16,Z 489.253,A -85,B 0,C 180,E1 -11003.574,E2 -11003.574} C_VEL
LIN {X 0,Y 404.175,Z 489.257,A -85,B 0,C 180,E1 -11005.766,E2 -11005.766} C_VEL
LIN {X 0,Y 404.189,Z 489.261,A -85,B 0,C 180,E1 -11007.999,E2 -11007.999} C_VEL
LIN {X 0,Y 404.137,Z 489.259,A -85,B 0,C 180,E1 -11011.56,E2 -11011.56} C_VEL
LIN {X 0,Y 404.177,Z 489.259,A -85,B 0,C 180,E1 -11015.016,E2 -11015.016} C_VEL
LIN {X 0,Y 404.151,Z 489.265,A -85,B 0,C 180,E1 -11018.757,E2 -11018.757} C_VEL
LIN {X 0,Y 404.18,Z 489.257,A -85,B 0,C 180,E1 -11021.61,E2 -11021.61} C_VEL
LIN {X 0,Y 404.194,Z 489.254,A -85,B 0,C 180,E1 -11024.53,E2 -11024.53} C_VEL
LIN {X 0,Y 404.199,Z 489.226,A -85,B 0,C 180,E1 -11027.305,E2 -11027.305} C_VEL
LIN {X 0,Y 404.164,Z 489.268,A -85,B 0,C 180,E1 -11029.956,E2 -11029.956} C_VEL
LIN {X 0,Y 404.134,Z 489.247,A -85,B 0,C 180,E1 -11033.124,E2 -11033.124} C_VEL
LIN {X 0,Y 404.139,Z 489.271,A -85,B 0,C 180,E1 -11036.188,E2 -11036.188} C_VEL
LIN {X 0,Y 404.148,Z 489.271,A -85,B 0,C 180,E1 -11039.716,E2 -11039.716} C_VEL
LIN {X 0,Y 404.19,Z 489.263,A -85,B 0,C 180,E1 -11043.123,E2 -11043.123} C_VEL
LIN {X 0,Y 404.172,Z 489.266,A -85,B 0,C 180,E1 -11045.335,E2 -11045.335} C_VEL
LIN {X 0,Y 404.134,Z 489.27,A -85,B 0,C 180,E1 -11048.581,E2 -11048.581} C_VEL
LIN {X 0,Y 404.206,Z 489.262,A -85,B 0,C 180,E1 -11051.762,E2 -11051.762} C_VEL
LIN {X 0,Y 404.202,Z 489.263,A -85,B 0,C 180,E1 -11054.882,E2 -11054.882} C_VEL
LIN {X 0,Y 404.252,Z 489.256,A -85,B 0,C 180,E1 -11057.959,E2 -11057.959} C_VEL
LIN {X 0,Y 404.429,Z 489.234,A -85,B 0,C 180,E1 -11062.1,E2 -11062.1} C_VEL
LIN {X 0,Y 404.42,Z 489.235,A -85,B 0,C 180,E1 -11064.015,E2 -11064.015} C_VEL
LIN {X 0,Y 404.479,Z 489.229,A -85,B 0,C 180,E1 -11068.009,E2 -11068.009} C_VEL
LIN {X 0,Y 404.608,Z 489.214,A -85,B 0,C 180,E1 -11070,E2 -11070} C_VEL
LIN {X 0,Y 404.419,Z 489.236,A -85,B 0,C 180,E1 -11072.988,E2 -11072.988} C_VEL
LIN {X 0,Y 404.408,Z 489.237,A -85,B 0,C 180,E1 -11076.987,E2 -11076.987} C_VEL
LIN {X 0,Y 404.254,Z 489.256,A -85,B 0,C 180,E1 -11080.012,E2 -11080.012} C_VEL
LIN {X 0,Y 404.262,Z 489.255,A -85,B 0,C 180,E1 -11083.211,E2 -11083.211} C_VEL
LIN {X 0,Y 404.211,Z 489.262,A -85,B 0,C 180,E1 -11087.007,E2 -11087.007} C_VEL
LIN {X 0,Y 404.159,Z 489.268,A -85,B 0,C 180,E1 -11090.351,E2 -11090.351} C_VEL
LIN {X 0,Y 404.131,Z 489.269,A -85,B 0,C 180,E1 -11091.928,E2 -11091.928} C_VEL
LIN {X 0,Y 403.489,Z 489.352,A -85,B 0,C 180,E1 -11092.76,E2 -11092.76} C_VEL
LIN {X 0,Y 400.656,Z 489.71,A -85,B 0,C 180,E1 -11094.112,E2 -11094.112} C_VEL
LIN {X 0,Y 398.246,Z 490.011,A -85,B 0,C 180,E1 -11095.204,E2 -11095.204} C_VEL
LIN {X 0,Y 397.212,Z 490.136,A -85,B 0,C 180,E1 -11096.048,E2 -11096.048} C_VEL
LIN {X 0,Y 397.129,Z 490.144,A -85,B 0,C 180,E1 -11096.334,E2 -11096.334} C_VEL
LIN {X 0,Y 397.121,Z 490.145,A -85,B 0,C 180,E1 -11098.543,E2 -11098.543} C_VEL
LIN {X 0,Y 397.075,Z 490.152,A -85,B 0,C 180,E1 -11102.071,E2 -11102.071} C_VEL
LIN {X 0,Y 397.114,Z 490.131,A -85,B 0,C 180,E1 -11105.503,E2 -11105.503} C_VEL
LIN {X 0,Y 397.131,Z 490.141,A -85,B 0,C 180,E1 -11108.863,E2 -11108.863} C_VEL
LIN {X 0,Y 397.151,Z 490.108,A -85,B 0,C 180,E1 -11112.255,E2 -11112.255} C_VEL
LIN {X 0,Y 397.143,Z 490.13,A -85,B 0,C 180,E1 -11115.059,E2 -11115.059} C_VEL
LIN {X 0,Y 397.147,Z 490.138,A -85,B 0,C 180,E1 -11118.007,E2 -11118.007} C_VEL
LIN {X 0,Y 397.099,Z 490.146,A -85,B 0,C 180,E1 -11121.725,E2 -11121.725} C_VEL
LIN {X 0,Y 397.117,Z 490.138,A -85,B 0,C 180,E1 -11125.507,E2 -11125.507} C_VEL
LIN {X 0,Y 397.077,Z 490.132,A -85,B 0,C 180,E1 -11129.118,E2 -11129.118} C_VEL
LIN {X 0,Y 397.186,Z 490.135,A -85,B 0,C 180,E1 -11132.61,E2 -11132.61} C_VEL
LIN {X 0,Y 397.124,Z 490.125,A -85,B 0,C 180,E1 -11135.982,E2 -11135.982} C_VEL
LIN {X 0,Y 397.13,Z 490.139,A -85,B 0,C 180,E1 -11139.705,E2 -11139.705} C_VEL
LIN {X 0,Y 397.173,Z 490.119,A -85,B 0,C 180,E1 -11142.845,E2 -11142.845} C_VEL
LIN {X 0,Y 397.22,Z 490.13,A -85,B 0,C 180,E1 -11146.703,E2 -11146.703} C_VEL
LIN {X 0,Y 397.209,Z 490.112,A -85,B 0,C 180,E1 -11149.809,E2 -11149.809} C_VEL
LIN {X 0,Y 397.343,Z 490.113,A -85,B 0,C 180,E1 -11152.888,E2 -11152.888} C_VEL
LIN {X 0,Y 397.253,Z 490.121,A -85,B 0,C 180,E1 -11154.926,E2 -11154.926} C_VEL
LIN {X 0,Y 397.443,Z 490.079,A -85,B 0,C 180,E1 -11157.974,E2 -11157.974} C_VEL
LIN {X 0,Y 397.572,Z 490.076,A -85,B 0,C 180,E1 -11160,E2 -11160} C_VEL
LIN {X 0,Y 397.374,Z 490.104,A -85,B 0,C 180,E1 -11163.042,E2 -11163.042} C_VEL
LIN {X 0,Y 397.367,Z 490.089,A -85,B 0,C 180,E1 -11166.092,E2 -11166.092} C_VEL
LIN {X 0,Y 397.245,Z 490.126,A -85,B 0,C 180,E1 -11169.162,E2 -11169.162} C_VEL
LIN {X 0,Y 397.211,Z 490.119,A -85,B 0,C 180,E1 -11172.259,E2 -11172.259} C_VEL
LIN {X 0,Y 397.171,Z 490.13,A -85,B 0,C 180,E1 -11175.393,E2 -11175.393} C_VEL
LIN {X 0,Y 397.155,Z 490.134,A -85,B 0,C 180,E1 -11178.574,E2 -11178.574} C_VEL
LIN {X 0,Y 397.089,Z 490.134,A -85,B 0,C 180,E1 -11181.819,E2 -11181.819} C_VEL
LIN {X 0,Y 397.147,Z 490.133,A -85,B 0,C 180,E1 -11185.513,E2 -11185.513} C_VEL
LIN {X 0,Y 397.116,Z 490.135,A -85,B 0,C 180,E1 -11188.545,E2 -11188.545} C_VEL
LIN {X 0,Y 397.073,Z 490.144,A -85,B 0,C 180,E1 -11192.072,E2 -11192.072} C_VEL
LIN {X 0,Y 397.116,Z 490.142,A -85,B 0,C 180,E1 -11195.504,E2 -11195.504} C_VEL
LIN {X 0,Y 397.133,Z 490.138,A -85,B 0,C 180,E1 -11198.864,E2 -11198.864} C_VEL
LIN {X 0,Y 397.11,Z 490.138,A -85,B 0,C 180,E1 -11202.262,E2 -11202.262} C_VEL
LIN {X 0,Y 397.086,Z 490.14,A -85,B 0,C 180,E1 -11205.069,E2 -11205.069} C_VEL
LIN {X 0,Y 397.066,Z 490.141,A -85,B 0,C 180,E1 -11208.022,E2 -11208.022} C_VEL
LIN {X 0,Y 397.13,Z 490.122,A -85,B 0,C 180,E1 -11211.139,E2 -11211.139} C_VEL
LIN {X 0,Y 397.118,Z 490.093,A -85,B 0,C 180,E1 -11214.498,E2 -11214.498} C_VEL
LIN {X 0,Y 397.162,Z 490.289,A -85,B 0,C 180,E1 -11217.487,E2 -11217.487} C_VEL
LIN {X 0,Y 399.146,Z 499.603,A -85,B 0,C 180,E1 -11220.097,E2 -11220.097} C_VEL
LIN {X 0,Y 401.038,Z 509.339,A -85,B 0,C 180,E1 -11222.612,E2 -11222.612} C_VEL
LIN {X 0,Y 400.551,Z 517.365,A -85,B 0,C 180,E1 -11224.541,E2 -11224.541} C_VEL
LIN {X 0,Y 400.149,Z 521.699,A -85,B 0,C 180,E1 -11225.559,E2 -11225.559} C_VEL
LIN {X 0,Y 401.429,Z 527.595,A -85,B 0,C 180,E1 -11225.801,E2 -11225.801} C_VEL
LIN {X 0,Y 407.072,Z 555.234,A -85,B 0,C 180,E1 -11226.674,E2 -11226.674} C_VEL
LIN {X 0,Y 407.143,Z 563.149,A -85,B 0,C 180,E1 -11226.827,E2 -11226.827} C_VEL
LIN {X 0,Y 405.541,Z 657.242,A -85,B 0,C 180,E1 -11228.526,E2 -11228.526} C_VEL
LIN {X 0,Y 405.053,Z 668.192,A -85,B 0,C 180,E1 -11228.832,E2 -11228.832} C_VEL
LIN {X 0,Y 404.43,Z 679.183,A -85,B 0,C 180,E1 -11229.264,E2 -11229.264} C_VEL
LIN {X 0,Y 403.787,Z 689.023,A -85,B 0,C 180,E1 -11229.765,E2 -11229.765} C_VEL
LIN {X 0,Y 402.989,Z 699.002,A -85,B 0,C 180,E1 -11230.388,E2 -11230.388} C_VEL
LIN {X 0,Y 402.184,Z 708.874,A -85,B 0,C 180,E1 -11231.139,E2 -11231.139} C_VEL
LIN {X 0,Y 401.215,Z 718.599,A -85,B 0,C 180,E1 -11232.018,E2 -11232.018} C_VEL
LIN {X 0,Y 400.218,Z 728.02,A -85,B 0,C 180,E1 -11233.026,E2 -11233.026} C_VEL
LIN {X 0,Y 399.316,Z 737.045,A -85,B 0,C 180,E1 -11234.169,E2 -11234.169} C_VEL
LIN {X 0,Y 398.594,Z 744.022,A -85,B 0,C 180,E1 -11235.187,E2 -11235.187} C_VEL
LIN {X 0,Y 397.902,Z 751.468,A -85,B 0,C 180,E1 -11236.45,E2 -11236.45} C_VEL
LIN {X 0,Y 397.319,Z 758.027,A -85,B 0,C 180,E1 -11237.745,E2 -11237.745} C_VEL
LIN {X 0,Y 396.664,Z 764.566,A -85,B 0,C 180,E1 -11239.279,E2 -11239.279} C_VEL
LIN {X 0,Y 396.282,Z 770,A -85,B 0,C 180,E1 -11240.816,E2 -11240.816} C_VEL
LIN {X 0,Y 396.006,Z 774.443,A -85,B 0,C 180,E1 -11242.351,E2 -11242.351} C_VEL
LIN {X 0,Y 395.862,Z 777.987,A -85,B 0,C 180,E1 -11243.885,E2 -11243.885} C_VEL
LIN {X 0,Y 395.803,Z 779.926,A -85,B 0,C 180,E1 -11244.907,E2 -11244.907} C_VEL
LIN {X 0,Y 395.723,Z 782.606,A -85,B 0,C 180,E1 -11246.946,E2 -11246.946} C_VEL
LIN {X 0,Y 395.79,Z 783.896,A -85,B 0,C 180,E1 -11248.983,E2 -11248.983} C_VEL
LIN {X 0,Y 395.777,Z 784.147,A -85,B 0,C 180,E1 -11250,E2 -11250} C_VEL
LIN {X 0,Y 395.761,Z 783.423,A -85,B 0,C 180,E1 -11252.035,E2 -11252.035} C_VEL
LIN {X 0,Y 395.722,Z 782.606,A -85,B 0,C 180,E1 -11253.054,E2 -11253.054} C_VEL
LIN {X 0,Y 395.8,Z 779.925,A -85,B 0,C 180,E1 -11255.093,E2 -11255.093} C_VEL
LIN {X 0,Y 395.925,Z 777.089,A -85,B 0,C 180,E1 -11256.574,E2 -11256.574} C_VEL
LIN {X 0,Y 396.075,Z 773.146,A -85,B 0,C 180,E1 -11258.161,E2 -11258.161} C_VEL
LIN {X 0,Y 396.389,Z 768.384,A -85,B 0,C 180,E1 -11259.697,E2 -11259.697} C_VEL
LIN {X 0,Y 396.993,Z 761.44,A -85,B 0,C 180,E1 -11261.488,E2 -11261.488} C_VEL
LIN {X 0,Y 397.482,Z 755.563,A -85,B 0,C 180,E1 -11262.768,E2 -11262.768} C_VEL
LIN {X 0,Y 398.265,Z 747.147,A -85,B 0,C 180,E1 -11264.303,E2 -11264.303} C_VEL
LIN {X 0,Y 398.934,Z 740.683,A -85,B 0,C 180,E1 -11265.322,E2 -11265.322} C_VEL
LIN {X 0,Y 399.896,Z 731.2,A -85,B 0,C 180,E1 -11266.594,E2 -11266.594} C_VEL
LIN {X 0,Y 400.849,Z 722.321,A -85,B 0,C 180,E1 -11267.604,E2 -11267.604} C_VEL
LIN {X 0,Y 401.802,Z 713.269,A -85,B 0,C 180,E1 -11268.483,E2 -11268.483} C_VEL
LIN {X 0,Y 402.747,Z 702.46,A -85,B 0,C 180,E1 -11269.363,E2 -11269.363} C_VEL
LIN {X 0,Y 403.543,Z 692.257,A -85,B 0,C 180,E1 -11270.048,E2 -11270.048} C_VEL
LIN {X 0,Y 404.229,Z 681.902,A -85,B 0,C 180,E1 -11270.613,E2 -11270.613} C_VEL
LIN {X 0,Y 404.944,Z 670.015,A -85,B 0,C 180,E1 -11271.107,E2 -11271.107} C_VEL
LIN {X 0,Y 405.468,Z 658.601,A -85,B 0,C 180,E1 -11271.445,E2 -11271.445} C_VEL
LIN {X 0,Y 406.127,Z 628.49,A -85,B 0,C 180,E1 -11272.009,E2 -11272.009} C_VEL
LIN {X 0,Y 407.207,Z 556.154,A -85,B 0,C 180,E1 -11273.3,E2 -11273.3} C_VEL
LIN {X 0,Y 401.438,Z 527.525,A -85,B 0,C 180,E1 -11274.2,E2 -11274.2} C_VEL
LIN {X 0,Y 400.18,Z 521.818,A -85,B 0,C 180,E1 -11274.424,E2 -11274.424} C_VEL
LIN {X 0,Y 401.152,Z 510.58,A -85,B 0,C 180,E1 -11277.097,E2 -11277.097} C_VEL
LIN {X 0,Y 399.764,Z 502.342,A -85,B 0,C 180,E1 -11279.236,E2 -11279.236} C_VEL
LIN {X 0,Y 397.162,Z 490.32,A -85,B 0,C 180,E1 -11282.513,E2 -11282.513} C_VEL
LIN {X 0,Y 397.106,Z 490.091,A -85,B 0,C 180,E1 -11285.734,E2 -11285.734} C_VEL
LIN {X 0,Y 397.112,Z 490.136,A -85,B 0,C 180,E1 -11289.576,E2 -11289.576} C_VEL
LIN {X 0,Y 397.102,Z 490.125,A -85,B 0,C 180,E1 -11293.478,E2 -11293.478} C_VEL
LIN {X 0,Y 397.101,Z 490.144,A -85,B 0,C 180,E1 -11296.52,E2 -11296.52} C_VEL
LIN {X 0,Y 397.116,Z 490.145,A -85,B 0,C 180,E1 -11299.551,E2 -11299.551} C_VEL
LIN {X 0,Y 397.094,Z 490.138,A -85,B 0,C 180,E1 -11302.789,E2 -11302.789} C_VEL
LIN {X 0,Y 397.114,Z 490.133,A -85,B 0,C 180,E1 -11306.281,E2 -11306.281} C_VEL
LIN {X 0,Y 397.099,Z 490.143,A -85,B 0,C 180,E1 -11310.135,E2 -11310.135} C_VEL
LIN {X 0,Y 397.188,Z 490.119,A -85,B 0,C 180,E1 -11312.609,E2 -11312.609} C_VEL
LIN {X 0,Y 397.123,Z 490.141,A -85,B 0,C 180,E1 -11315.981,E2 -11315.981} C_VEL
LIN {X 0,Y 397.132,Z 490.126,A -85,B 0,C 180,E1 -11319.704,E2 -11319.704} C_VEL
LIN {X 0,Y 397.175,Z 490.134,A -85,B 0,C 180,E1 -11322.844,E2 -11322.844} C_VEL
LIN {X 0,Y 397.221,Z 490.107,A -85,B 0,C 180,E1 -11326.702,E2 -11326.702} C_VEL
LIN {X 0,Y 397.21,Z 490.132,A -85,B 0,C 180,E1 -11329.808,E2 -11329.808} C_VEL
LIN {X 0,Y 397.348,Z 490.105,A -85,B 0,C 180,E1 -11332.887,E2 -11332.887} C_VEL
LIN {X 0,Y 397.248,Z 490.104,A -85,B 0,C 180,E1 -11334.925,E2 -11334.925} C_VEL
LIN {X 0,Y 397.443,Z 490.1,A -85,B 0,C 180,E1 -11337.973,E2 -11337.973} C_VEL
LIN {X 0,Y 397.572,Z 490.076,A -85,B 0,C 180,E1 -11340,E2 -11340} C_VEL
LIN {X 0,Y 397.374,Z 490.09,A -85,B 0,C 180,E1 -11343.041,E2 -11343.041} C_VEL
LIN {X 0,Y 397.338,Z 490.111,A -85,B 0,C 180,E1 -11346.653,E2 -11346.653} C_VEL
LIN {X 0,Y 397.244,Z 490.111,A -85,B 0,C 180,E1 -11349.162,E2 -11349.162} C_VEL
LIN {X 0,Y 397.21,Z 490.128,A -85,B 0,C 180,E1 -11352.258,E2 -11352.258} C_VEL
LIN {X 0,Y 397.17,Z 490.132,A -85,B 0,C 180,E1 -11355.392,E2 -11355.392} C_VEL
LIN {X 0,Y 397.153,Z 490.127,A -85,B 0,C 180,E1 -11358.573,E2 -11358.573} C_VEL
LIN {X 0,Y 397.1,Z 490.143,A -85,B 0,C 180,E1 -11361.818,E2 -11361.818} C_VEL
LIN {X 0,Y 397.144,Z 490.128,A -85,B 0,C 180,E1 -11365.512,E2 -11365.512} C_VEL
LIN {X 0,Y 397.118,Z 490.138,A -85,B 0,C 180,E1 -11368.543,E2 -11368.543} C_VEL
LIN {X 0,Y 397.102,Z 490.143,A -85,B 0,C 180,E1 -11372.069,E2 -11372.069} C_VEL
LIN {X 0,Y 397.112,Z 490.135,A -85,B 0,C 180,E1 -11375.504,E2 -11375.504} C_VEL
LIN {X 0,Y 397.126,Z 490.141,A -85,B 0,C 180,E1 -11378.862,E2 -11378.862} C_VEL
LIN {X 0,Y 397.151,Z 490.139,A -85,B 0,C 180,E1 -11382.256,E2 -11382.256} C_VEL
LIN {X 0,Y 397.143,Z 490.127,A -85,B 0,C 180,E1 -11385.06,E2 -11385.06} C_VEL
LIN {X 0,Y 397.149,Z 490.112,A -85,B 0,C 180,E1 -11388.007,E2 -11388.007} C_VEL
LIN {X 0,Y 397.104,Z 490.134,A -85,B 0,C 180,E1 -11391.726,E2 -11391.726} C_VEL
LIN {X 0,Y 397.12,Z 490.142,A -85,B 0,C 180,E1 -11395.507,E2 -11395.507} C_VEL
LIN {X 0,Y 397.079,Z 490.149,A -85,B 0,C 180,E1 -11399.118,E2 -11399.118} C_VEL
LIN {X 0,Y 397.189,Z 490.135,A -85,B 0,C 180,E1 -11402.61,E2 -11402.61} C_VEL
LIN {X 0,Y 397.128,Z 490.144,A -85,B 0,C 180,E1 -11405.982,E2 -11405.982} C_VEL
LIN {X 0,Y 397.134,Z 490.143,A -85,B 0,C 180,E1 -11409.705,E2 -11409.705} C_VEL
LIN {X 0,Y 397.177,Z 490.138,A -85,B 0,C 180,E1 -11412.845,E2 -11412.845} C_VEL
LIN {X 0,Y 397.224,Z 490.132,A -85,B 0,C 180,E1 -11416.703,E2 -11416.703} C_VEL
LIN {X 0,Y 397.214,Z 490.133,A -85,B 0,C 180,E1 -11419.809,E2 -11419.809} C_VEL
LIN {X 0,Y 397.36,Z 490.114,A -85,B 0,C 180,E1 -11422.888,E2 -11422.888} C_VEL
LIN {X 0,Y 397.252,Z 490.133,A -85,B 0,C 180,E1 -11424.925,E2 -11424.925} C_VEL
LIN {X 0,Y 397.476,Z 490.393,A -85,B 0,C 180,E1 -11427.973,E2 -11427.973} C_VEL
LIN {X 0,Y 397.65,Z 490.5,A -85,B 0,C 180,E1 -11430,E2 -11430} C_VEL
LIN {X 0,Y 397.378,Z 490.263,A -85,B 0,C 180,E1 -11433.041,E2 -11433.041} C_VEL
LIN {X 0,Y 397.36,Z 490.115,A -85,B 0,C 180,E1 -11437.112,E2 -11437.112} C_VEL
LIN {X 0,Y 397.214,Z 490.133,A -85,B 0,C 180,E1 -11440.191,E2 -11440.191} C_VEL
LIN {X 0,Y 397.222,Z 490.133,A -85,B 0,C 180,E1 -11443.321,E2 -11443.321} C_VEL
LIN {X 0,Y 397.177,Z 490.138,A -85,B 0,C 180,E1 -11447.155,E2 -11447.155} C_VEL
LIN {X 0,Y 397.098,Z 490.148,A -85,B 0,C 180,E1 -11450.73,E2 -11450.73} C_VEL
LIN {X 0,Y 397.128,Z 490.144,A -85,B 0,C 180,E1 -11454.018,E2 -11454.018} C_VEL
LIN {X 0,Y 397.129,Z 490.144,A -85,B 0,C 180,E1 -11456.334,E2 -11456.334} C_VEL
LIN {X 0,Y 396.46,Z 490.226,A -85,B 0,C 180,E1 -11457.181,E2 -11457.181} C_VEL
LIN {X 0,Y 393.587,Z 490.585,A -85,B 0,C 180,E1 -11458.556,E2 -11458.556} C_VEL
LIN {X 0,Y 391.15,Z 490.889,A -85,B 0,C 180,E1 -11459.668,E2 -11459.668} C_VEL
LIN {X 0,Y 390.098,Z 491.02,A -85,B 0,C 180,E1 -11460.528,E2 -11460.528} C_VEL
LIN {X 0,Y 390.01,Z 491.028,A -85,B 0,C 180,E1 -11460.819,E2 -11460.819} C_VEL
LIN {X 0,Y 390.062,Z 491.025,A -85,B 0,C 180,E1 -11464.024,E2 -11464.024} C_VEL
LIN {X 0,Y 390.041,Z 491.005,A -85,B 0,C 180,E1 -11467.551,E2 -11467.551} C_VEL
LIN {X 0,Y 390.076,Z 491.014,A -85,B 0,C 180,E1 -11470.826,E2 -11470.826} C_VEL
